LIN {X 0,Y 328.389,Z 347.877,A -85,B 0,C 180,E1 -14879.488,E2 -14879.488} C_VEL
LIN {X 0,Y 329.533,Z 341.284,A -85,B 0,C 180,E1 -14882.946,E2 -14882.946} C_VEL
LIN {X 0,Y 330.904,Z 335.131,A -85,B 0,C 180,E1 -14886.49,E2 -14886.49} C_VEL
LIN {X 0,Y 331.138,Z 332.463,A -85,B 0,C 180,E1 -14888.253,E2 -14888.253} C_VEL
LIN {X 0,Y 330.484,Z 328.715,A -85,B 0,C 180,E1 -14891.242,E2 -14891.242} C_VEL
LIN {X 0,Y 329.857,Z 325.225,A -85,B 0,C 180,E1 -14894.677,E2 -14894.677} C_VEL
LIN {X 0,Y 329.364,Z 322.49,A -85,B 0,C 180,E1 -14898.317,E2 -14898.317} C_VEL
LIN {X 0,Y 329.011,Z 320.792,A -85,B 0,C 180,E1 -14901.723,E2 -14901.723} C_VEL
LIN {X 0,Y 328.795,Z 319.94,A -85,B 0,C 180,E1 -14904.751,E2 -14904.751} C_VEL
LIN {X 0,Y 328.622,Z 319.641,A -85,B 0,C 180,E1 -14907.679,E2 -14907.679} C_VEL
LIN {X 0,Y 328.631,Z 319.835,A -85,B 0,C 180,E1 -14911.261,E2 -14911.261} C_VEL
LIN {X 0,Y 328.579,Z 320.736,A -85,B 0,C 180,E1 -14914.803,E2 -14914.803} C_VEL
LIN {X 0,Y 329.786,Z 323.377,A -85,B 0,C 180,E1 -14915.189,E2 -14915.189} C_VEL
LIN {X 0,Y 331.608,Z 326.284,A -85,B 0,C 180,E1 -14915.69,E2 -14915.69} C_VEL
LIN {X 0,Y 336.582,Z 336.57,A -85,B 0,C 180,E1 -14917.291,E2 -14917.291} C_VEL
LIN {X 0,Y 339.409,Z 344.725,A -85,B 0,C 180,E1 -14918.474,E2 -14918.474} C_VEL
LIN {X 0,Y 339.579,Z 346.937,A -85,B 0,C 180,E1 -14918.735,E2 -14918.735} C_VEL
LIN {X 0,Y 338.027,Z 357.85,A -85,B 0,C 180,E1 -14919.853,E2 -14919.853} C_VEL
LIN {X 0,Y 336.397,Z 367.772,A -85,B 0,C 180,E1 -14921.106,E2 -14921.106} C_VEL
LIN {X 0,Y 334.71,Z 377.405,A -85,B 0,C 180,E1 -14922.59,E2 -14922.59} C_VEL
LIN {X 0,Y 333.131,Z 385.421,A -85,B 0,C 180,E1 -14924.082,E2 -14924.082} C_VEL
LIN {X 0,Y 331.535,Z 393.277,A -85,B 0,C 180,E1 -14925.89,E2 -14925.89} C_VEL
LIN {X 0,Y 330.035,Z 399.65,A -85,B 0,C 180,E1 -14927.705,E2 -14927.705} C_VEL
LIN {X 0,Y 328.96,Z 404.549,A -85,B 0,C 180,E1 -14929.49,E2 -14929.49} C_VEL
LIN {X 0,Y 327.87,Z 408.533,A -85,B 0,C 180,E1 -14931.37,E2 -14931.37} C_VEL
LIN {X 0,Y 327.396,Z 410.536,A -85,B 0,C 180,E1 -14932.6,E2 -14932.6} C_VEL
LIN {X 0,Y 326.97,Z 412.06,A -85,B 0,C 180,E1 -14933.83,E2 -14933.83} C_VEL
LIN {X 0,Y 326.554,Z 413.149,A -85,B 0,C 180,E1 -14935.062,E2 -14935.062} C_VEL
LIN {X 0,Y 326.145,Z 413.838,A -85,B 0,C 180,E1 -14936.294,E2 -14936.294} C_VEL
LIN {X 0,Y 325.84,Z 414.097,A -85,B 0,C 180,E1 -14937.528,E2 -14937.528} C_VEL
LIN {X 0,Y 325.67,Z 413.896,A -85,B 0,C 180,E1 -14938.764,E2 -14938.764} C_VEL
LIN {X 0,Y 325.61,Z 413.286,A -85,B 0,C 180,E1 -14940,E2 -14940} C_VEL
LIN {X 0,Y 325.631,Z 412.265,A -85,B 0,C 180,E1 -14941.237,E2 -14941.237} C_VEL
LIN {X 0,Y 325.654,Z 410.778,A -85,B 0,C 180,E1 -14942.474,E2 -14942.474} C_VEL
LIN {X 0,Y 325.946,Z 407.724,A -85,B 0,C 180,E1 -14944.328,E2 -14944.328} C_VEL
LIN {X 0,Y 326.069,Z 403.613,A -85,B 0,C 180,E1 -14946.187,E2 -14946.187} C_VEL
LIN {X 0,Y 326.438,Z 397.331,A -85,B 0,C 180,E1 -14948.356,E2 -14948.356} C_VEL
LIN {X 0,Y 326.972,Z 390.471,A -85,B 0,C 180,E1 -14950.214,E2 -14950.214} C_VEL
LIN {X 0,Y 327.683,Z 381.942,A -85,B 0,C 180,E1 -14952.071,E2 -14952.071} C_VEL
LIN {X 0,Y 328.388,Z 373.312,A -85,B 0,C 180,E1 -14953.616,E2 -14953.616} C_VEL
LIN {X 0,Y 329.324,Z 362.847,A -85,B 0,C 180,E1 -14955.155,E2 -14955.155} C_VEL
LIN {X 0,Y 330.164,Z 350.596,A -85,B 0,C 180,E1 -14956.613,E2 -14956.613} C_VEL
LIN {X 0,Y 330.93,Z 338.24,A -85,B 0,C 180,E1 -14957.775,E2 -14957.775} C_VEL
LIN {X 0,Y 331.318,Z 331.336,A -85,B 0,C 180,E1 -14958.313,E2 -14958.313} C_VEL
LIN {X 0,Y 328.408,Z 318.06,A -85,B 0,C 180,E1 -14959.286,E2 -14959.286} C_VEL
LIN {X 0,Y 326.112,Z 308.863,A -85,B 0,C 180,E1 -14959.869,E2 -14959.869} C_VEL
LIN {X 0,Y 326.351,Z 308.833,A -85,B 0,C 180,E1 -14962.807,E2 -14962.807} C_VEL
LIN {X 0,Y 326.567,Z 308.8,A -85,B 0,C 180,E1 -14965.494,E2 -14965.494} C_VEL
LIN {X 0,Y 326.634,Z 308.796,A -85,B 0,C 180,E1 -14968.253,E2 -14968.253} C_VEL
LIN {X 0,Y 326.592,Z 308.795,A -85,B 0,C 180,E1 -14971.095,E2 -14971.095} C_VEL
LIN {X 0,Y 326.61,Z 308.804,A -85,B 0,C 180,E1 -14974.019,E2 -14974.019} C_VEL
LIN {X 0,Y 326.63,Z 308.801,A -85,B 0,C 180,E1 -14977.239,E2 -14977.239} C_VEL
LIN {X 0,Y 326.58,Z 308.807,A -85,B 0,C 180,E1 -14981.131,E2 -14981.131} C_VEL
LIN {X 0,Y 326.53,Z 308.809,A -85,B 0,C 180,E1 -14984.743,E2 -14984.743} C_VEL
LIN {X 0,Y 326.578,Z 308.805,A -85,B 0,C 180,E1 -14988.154,E2 -14988.154} C_VEL
LIN {X 0,Y 326.598,Z 308.804,A -85,B 0,C 180,E1 -14991.388,E2 -14991.388} C_VEL
LIN {X 0,Y 326.571,Z 308.814,A -85,B 0,C 180,E1 -14994.598,E2 -14994.598} C_VEL
LIN {X 0,Y 326.816,Z 310.846,A -85,B 0,C 180,E1 -14996.005,E2 -14996.005} C_VEL
LIN {X 0,Y 326.471,Z 317.34,A -85,B 0,C 180,E1 -15000.322,E2 -15000.322} C_VEL
LIN {X 0,Y 326.342,Z 322.733,A -85,B 0,C 180,E1 -15003.801,E2 -15003.801} C_VEL
LIN {X 0,Y 326.339,Z 329.269,A -85,B 0,C 180,E1 -15007.772,E2 -15007.772} C_VEL
LIN {X 0,Y 330.703,Z 344.202,A -85,B 0,C 180,E1 -15008.694,E2 -15008.694} C_VEL
LIN {X 0,Y 333.363,Z 356.048,A -85,B 0,C 180,E1 -15009.607,E2 -15009.607} C_VEL
LIN {X 0,Y 334.3,Z 361.022,A -85,B 0,C 180,E1 -15010.049,E2 -15010.049} C_VEL
LIN {X 0,Y 333.305,Z 372.846,A -85,B 0,C 180,E1 -15011.083,E2 -15011.083} C_VEL
LIN {X 0,Y 332.083,Z 384.217,A -85,B 0,C 180,E1 -15012.355,E2 -15012.355} C_VEL
LIN {X 0,Y 331.074,Z 393.497,A -85,B 0,C 180,E1 -15013.664,E2 -15013.664} C_VEL
LIN {X 0,Y 329.738,Z 402.364,A -85,B 0,C 180,E1 -15015.181,E2 -15015.181} C_VEL
LIN {X 0,Y 328.555,Z 410.995,A -85,B 0,C 180,E1 -15017.02,E2 -15017.02} C_VEL
LIN {X 0,Y 327.501,Z 417.914,A -85,B 0,C 180,E1 -15018.864,E2 -15018.864} C_VEL
LIN {X 0,Y 326.701,Z 423.408,A -85,B 0,C 180,E1 -15020.715,E2 -15020.715} C_VEL
LIN {X 0,Y 326.02,Z 428.45,A -85,B 0,C 180,E1 -15022.946,E2 -15022.946} C_VEL
LIN {X 0,Y 325.518,Z 431.838,A -85,B 0,C 180,E1 -15025.046,E2 -15025.046} C_VEL
LIN {X 0,Y 325.427,Z 433.241,A -85,B 0,C 180,E1 -15026.285,E2 -15026.285} C_VEL
LIN {X 0,Y 325.344,Z 434.228,A -85,B 0,C 180,E1 -15027.524,E2 -15027.524} C_VEL
LIN {X 0,Y 325.209,Z 435.072,A -85,B 0,C 180,E1 -15030,E2 -15030} C_VEL
LIN {X 0,Y 325.34,Z 434.294,A -85,B 0,C 180,E1 -15032.476,E2 -15032.476} C_VEL
LIN {X 0,Y 325.404,Z 433.335,A -85,B 0,C 180,E1 -15033.715,E2 -15033.715} C_VEL
LIN {X 0,Y 325.498,Z 431.982,A -85,B 0,C 180,E1 -15034.955,E2 -15034.955} C_VEL
LIN {X 0,Y 325.994,Z 428.727,A -85,B 0,C 180,E1 -15037.017,E2 -15037.017} C_VEL
LIN {X 0,Y 326.626,Z 423.679,A -85,B 0,C 180,E1 -15039.287,E2 -15039.287} C_VEL
LIN {X 0,Y 327.463,Z 418.244,A -85,B 0,C 180,E1 -15041.137,E2 -15041.137} C_VEL
LIN {X 0,Y 328.501,Z 411.435,A -85,B 0,C 180,E1 -15042.982,E2 -15042.982} C_VEL
LIN {X 0,Y 329.698,Z 402.902,A -85,B 0,C 180,E1 -15044.821,E2 -15044.821} C_VEL
LIN {X 0,Y 331.04,Z 394.145,A -85,B 0,C 180,E1 -15046.338,E2 -15046.338} C_VEL
LIN {X 0,Y 332.114,Z 384.041,A -85,B 0,C 180,E1 -15047.774,E2 -15047.774} C_VEL
LIN {X 0,Y 333.36,Z 372.347,A -85,B 0,C 180,E1 -15049.073,E2 -15049.073} C_VEL
LIN {X 0,Y 334.401,Z 361.794,A -85,B 0,C 180,E1 -15049.987,E2 -15049.987} C_VEL
LIN {X 0,Y 332.363,Z 351.218,A -85,B 0,C 180,E1 -15050.895,E2 -15050.895} C_VEL
LIN {X 0,Y 329.213,Z 338.732,A -85,B 0,C 180,E1 -15051.777,E2 -15051.777} C_VEL
LIN {X 0,Y 326.37,Z 329.318,A -85,B 0,C 180,E1 -15052.32,E2 -15052.32} C_VEL
LIN {X 0,Y 326.345,Z 322.926,A -85,B 0,C 180,E1 -15056.198,E2 -15056.198} C_VEL
LIN {X 0,Y 326.48,Z 317.517,A -85,B 0,C 180,E1 -15059.677,E2 -15059.677} C_VEL
LIN {X 0,Y 326.824,Z 311.012,A -85,B 0,C 180,E1 -15063.994,E2 -15063.994} C_VEL
LIN {X 0,Y 326.594,Z 308.806,A -85,B 0,C 180,E1 -15065.522,E2 -15065.522} C_VEL
LIN {X 0,Y 326.613,Z 308.802,A -85,B 0,C 180,E1 -15069.227,E2 -15069.227} C_VEL
LIN {X 0,Y 326.578,Z 308.809,A -85,B 0,C 180,E1 -15072.972,E2 -15072.972} C_VEL
LIN {X 0,Y 326.578,Z 308.807,A -85,B 0,C 180,E1 -15077.028,E2 -15077.028} C_VEL
LIN {X 0,Y 326.612,Z 308.801,A -85,B 0,C 180,E1 -15080.773,E2 -15080.773} C_VEL
LIN {X 0,Y 326.528,Z 308.807,A -85,B 0,C 180,E1 -15083.972,E2 -15083.972} C_VEL
LIN {X 0,Y 325.824,Z 309.013,A -85,B 0,C 180,E1 -15084.998,E2 -15084.998} C_VEL
LIN {X 0,Y 324.191,Z 309.573,A -85,B 0,C 180,E1 -15086,E2 -15086} C_VEL
LIN {X 0,Y 320.337,Z 311.597,A -85,B 0,C 180,E1 -15087.986,E2 -15087.986} C_VEL
LIN {X 0,Y 319.2,Z 313.002,A -85,B 0,C 180,E1 -15089.007,E2 -15089.007} C_VEL
LIN {X 0,Y 319.08,Z 313.52,A -85,B 0,C 180,E1 -15089.351,E2 -15089.351} C_VEL
LIN {X 0,Y 318.923,Z 319.269,A -85,B 0,C 180,E1 -15093.144,E2 -15093.144} C_VEL
LIN {X 0,Y 318.828,Z 324.595,A -85,B 0,C 180,E1 -15096.623,E2 -15096.623} C_VEL
LIN {X 0,Y 318.728,Z 329.745,A -85,B 0,C 180,E1 -15099.955,E2 -15099.955} C_VEL
LIN {X 0,Y 321.159,Z 342.779,A -85,B 0,C 180,E1 -15100.685,E2 -15100.685} C_VEL
LIN {X 0,Y 323.621,Z 355.679,A -85,B 0,C 180,E1 -15101.649,E2 -15101.649} C_VEL
LIN {X 0,Y 323.48,Z 361.623,A -85,B 0,C 180,E1 -15102.129,E2 -15102.129} C_VEL
LIN {X 0,Y 322.624,Z 373.758,A -85,B 0,C 180,E1 -15103.285,E2 -15103.285} C_VEL
LIN {X 0,Y 321.819,Z 385.197,A -85,B 0,C 180,E1 -15104.652,E2 -15104.652} C_VEL
LIN {X 0,Y 320.97,Z 394.854,A -85,B 0,C 180,E1 -15106.063,E2 -15106.063} C_VEL
LIN {X 0,Y 320.061,Z 405.398,A -85,B 0,C 180,E1 -15107.959,E2 -15107.959} C_VEL
LIN {X 0,Y 319.336,Z 413.85,A -85,B 0,C 180,E1 -15109.859,E2 -15109.859} C_VEL
LIN {X 0,Y 318.801,Z 420.704,A -85,B 0,C 180,E1 -15111.761,E2 -15111.761} C_VEL
LIN {X 0,Y 318.416,Z 426.181,A -85,B 0,C 180,E1 -15113.664,E2 -15113.664} C_VEL
LIN {X 0,Y 318.282,Z 430.405,A -85,B 0,C 180,E1 -15115.567,E2 -15115.567} C_VEL
LIN {X 0,Y 318.126,Z 433.53,A -85,B 0,C 180,E1 -15117.468,E2 -15117.468} C_VEL
LIN {X 0,Y 318.112,Z 435.035,A -85,B 0,C 180,E1 -15118.734,E2 -15118.734} C_VEL
LIN {X 0,Y 318.172,Z 436.12,A -85,B 0,C 180,E1 -15120,E2 -15120} C_VEL
LIN {X 0,Y 318.254,Z 436.733,A -85,B 0,C 180,E1 -15121.265,E2 -15121.265} C_VEL
LIN {X 0,Y 318.421,Z 436.924,A -85,B 0,C 180,E1 -15122.53,E2 -15122.53} C_VEL
LIN {X 0,Y 318.669,Z 436.708,A -85,B 0,C 180,E1 -15123.794,E2 -15123.794} C_VEL
LIN {X 0,Y 318.948,Z 436.024,A -85,B 0,C 180,E1 -15125.057,E2 -15125.057} C_VEL
LIN {X 0,Y 319.369,Z 433.443,A -85,B 0,C 180,E1 -15127.587,E2 -15127.587} C_VEL
LIN {X 0,Y 320.376,Z 430.263,A -85,B 0,C 180,E1 -15129.47,E2 -15129.47} C_VEL
LIN {X 0,Y 321.316,Z 425.996,A -85,B 0,C 180,E1 -15131.353,E2 -15131.353} C_VEL
LIN {X 0,Y 322.763,Z 419.488,A -85,B 0,C 180,E1 -15133.537,E2 -15133.537} C_VEL
LIN {X 0,Y 324.353,Z 412.416,A -85,B 0,C 180,E1 -15135.392,E2 -15135.392} C_VEL
LIN {X 0,Y 326.182,Z 403.606,A -85,B 0,C 180,E1 -15137.233,E2 -15137.233} C_VEL
LIN {X 0,Y 328.209,Z 393.435,A -85,B 0,C 180,E1 -15138.95,E2 -15138.95} C_VEL
LIN {X 0,Y 330.118,Z 382.681,A -85,B 0,C 180,E1 -15140.419,E2 -15140.419} C_VEL
LIN {X 0,Y 332.217,Z 369.516,A -85,B 0,C 180,E1 -15141.838,E2 -15141.838} C_VEL
LIN {X 0,Y 332.351,Z 368.078,A -85,B 0,C 180,E1 -15141.981,E2 -15141.981} C_VEL
LIN {X 0,Y 330.162,Z 358.055,A -85,B 0,C 180,E1 -15143.305,E2 -15143.305} C_VEL
LIN {X 0,Y 326.236,Z 347.061,A -85,B 0,C 180,E1 -15144.856,E2 -15144.856} C_VEL
LIN {X 0,Y 323.056,Z 340.093,A -85,B 0,C 180,E1 -15145.906,E2 -15145.906} C_VEL
LIN {X 0,Y 321.796,Z 337.014,A -85,B 0,C 180,E1 -15146.354,E2 -15146.354} C_VEL
LIN {X 0,Y 322.533,Z 332.112,A -85,B 0,C 180,E1 -15150.078,E2 -15150.078} C_VEL
LIN {X 0,Y 323.218,Z 328.529,A -85,B 0,C 180,E1 -15152.929,E2 -15152.929} C_VEL
LIN {X 0,Y 323.383,Z 326.836,A -85,B 0,C 180,E1 -15154.406,E2 -15154.406} C_VEL
LIN {X 0,Y 323.298,Z 324.738,A -85,B 0,C 180,E1 -15156.455,E2 -15156.455} C_VEL
LIN {X 0,Y 323.004,Z 322.421,A -85,B 0,C 180,E1 -15159.123,E2 -15159.123} C_VEL
LIN {X 0,Y 322.6,Z 320.404,A -85,B 0,C 180,E1 -15162.208,E2 -15162.208} C_VEL
LIN {X 0,Y 322.049,Z 319.739,A -85,B 0,C 180,E1 -15164.293,E2 -15164.293} C_VEL
LIN {X 0,Y 321.458,Z 319.688,A -85,B 0,C 180,E1 -15166.547,E2 -15166.547} C_VEL
LIN {X 0,Y 322.812,Z 326.631,A -85,B 0,C 180,E1 -15170.285,E2 -15170.285} C_VEL
LIN {X 0,Y 323.47,Z 330.981,A -85,B 0,C 180,E1 -15172.529,E2 -15172.529} C_VEL
LIN {X 0,Y 322.945,Z 335.629,A -85,B 0,C 180,E1 -15174.781,E2 -15174.781} C_VEL
LIN {X 0,Y 321.872,Z 343.274,A -85,B 0,C 180,E1 -15178.397,E2 -15178.397} C_VEL
LIN {X 0,Y 320.746,Z 352.365,A -85,B 0,C 180,E1 -15182.604,E2 -15182.604} C_VEL
LIN {X 0,Y 320.405,Z 355.766,A -85,B 0,C 180,E1 -15184.07,E2 -15184.07} C_VEL
LIN {X 0,Y 321.285,Z 359.893,A -85,B 0,C 180,E1 -15184.469,E2 -15184.469} C_VEL
LIN {X 0,Y 321.976,Z 362.193,A -85,B 0,C 180,E1 -15184.716,E2 -15184.716} C_VEL
LIN {X 0,Y 324.913,Z 374.79,A -85,B 0,C 180,E1 -15185.952,E2 -15185.952} C_VEL
LIN {X 0,Y 326.631,Z 386.508,A -85,B 0,C 180,E1 -15187.1,E2 -15187.1} C_VEL
LIN {X 0,Y 326.814,Z 401.047,A -85,B 0,C 180,E1 -15188.557,E2 -15188.557} C_VEL
LIN {X 0,Y 326.653,Z 413.267,A -85,B 0,C 180,E1 -15190.028,E2 -15190.028} C_VEL
LIN {X 0,Y 324.612,Z 424.833,A -85,B 0,C 180,E1 -15191.54,E2 -15191.54} C_VEL
LIN {X 0,Y 322.759,Z 435.331,A -85,B 0,C 180,E1 -15193.264,E2 -15193.264} C_VEL
LIN {X 0,Y 321.272,Z 444.462,A -85,B 0,C 180,E1 -15195.106,E2 -15195.106} C_VEL
LIN {X 0,Y 320.021,Z 452.055,A -85,B 0,C 180,E1 -15196.991,E2 -15196.991} C_VEL
LIN {X 0,Y 319.016,Z 459.185,A -85,B 0,C 180,E1 -15199.207,E2 -15199.207} C_VEL
LIN {X 0,Y 318.414,Z 464.012,A -85,B 0,C 180,E1 -15201.112,E2 -15201.112} C_VEL
LIN {X 0,Y 318.142,Z 467.739,A -85,B 0,C 180,E1 -15203.021,E2 -15203.021} C_VEL
LIN {X 0,Y 317.959,Z 470.454,A -85,B 0,C 180,E1 -15204.928,E2 -15204.928} C_VEL
LIN {X 0,Y 317.981,Z 471.724,A -85,B 0,C 180,E1 -15206.198,E2 -15206.198} C_VEL
LIN {X 0,Y 318.095,Z 472.979,A -85,B 0,C 180,E1 -15208.734,E2 -15208.734} C_VEL
LIN {X 0,Y 318.215,Z 472.983,A -85,B 0,C 180,E1 -15210,E2 -15210} C_VEL
LIN {X 0,Y 317.968,Z 471.876,A -85,B 0,C 180,E1 -15212.534,E2 -15212.534} C_VEL
LIN {X 0,Y 317.985,Z 470.852,A -85,B 0,C 180,E1 -15213.802,E2 -15213.802} C_VEL
LIN {X 0,Y 318.114,Z 467.745,A -85,B 0,C 180,E1 -15216.187,E2 -15216.187} C_VEL
LIN {X 0,Y 318.273,Z 463.753,A -85,B 0,C 180,E1 -15218.252,E2 -15218.252} C_VEL
LIN {X 0,Y 318.728,Z 458.888,A -85,B 0,C 180,E1 -15220.16,E2 -15220.16} C_VEL
LIN {X 0,Y 319.953,Z 449.69,A -85,B 0,C 180,E1 -15223.012,E2 -15223.012} C_VEL
LIN {X 0,Y 321.346,Z 440.86,A -85,B 0,C 180,E1 -15225.215,E2 -15225.215} C_VEL
LIN {X 0,Y 322.877,Z 431.604,A -85,B 0,C 180,E1 -15227.089,E2 -15227.089} C_VEL
LIN {X 0,Y 325.018,Z 420.298,A -85,B 0,C 180,E1 -15228.926,E2 -15228.926} C_VEL
LIN {X 0,Y 326.586,Z 411.332,A -85,B 0,C 180,E1 -15230.14,E2 -15230.14} C_VEL
LIN {X 0,Y 326.871,Z 400.124,A -85,B 0,C 180,E1 -15231.564,E2 -15231.564} C_VEL
LIN {X 0,Y 326.921,Z 389.197,A -85,B 0,C 180,E1 -15232.765,E2 -15232.765} C_VEL
LIN {X 0,Y 325.801,Z 378.126,A -85,B 0,C 180,E1 -15233.943,E2 -15233.943} C_VEL
LIN {X 0,Y 323.834,Z 367.884,A -85,B 0,C 180,E1 -15235.031,E2 -15235.031} C_VEL
LIN {X 0,Y 321.496,Z 359.207,A -85,B 0,C 180,E1 -15235.986,E2 -15235.986} C_VEL
LIN {X 0,Y 320.514,Z 355.252,A -85,B 0,C 180,E1 -15236.422,E2 -15236.422} C_VEL
LIN {X 0,Y 321.598,Z 347.856,A -85,B 0,C 180,E1 -15240.174,E2 -15240.174} C_VEL
LIN {X 0,Y 322.769,Z 341.576,A -85,B 0,C 180,E1 -15243.617,E2 -15243.617} C_VEL
LIN {X 0,Y 323.987,Z 336.568,A -85,B 0,C 180,E1 -15246.62,E2 -15246.62} C_VEL
LIN {X 0,Y 324.144,Z 333.59,A -85,B 0,C 180,E1 -15248.689,E2 -15248.689} C_VEL
LIN {X 0,Y 323.757,Z 331.199,A -85,B 0,C 180,E1 -15250.635,E2 -15250.635} C_VEL
LIN {X 0,Y 323.088,Z 327.59,A -85,B 0,C 180,E1 -15254.124,E2 -15254.124} C_VEL
LIN {X 0,Y 322.546,Z 324.723,A -85,B 0,C 180,E1 -15257.803,E2 -15257.803} C_VEL
LIN {X 0,Y 322.233,Z 323.095,A -85,B 0,C 180,E1 -15260.765,E2 -15260.765} C_VEL
LIN {X 0,Y 321.983,Z 322.01,A -85,B 0,C 180,E1 -15263.89,E2 -15263.89} C_VEL
LIN {X 0,Y 321.799,Z 321.521,A -85,B 0,C 180,E1 -15266.907,E2 -15266.907} C_VEL
LIN {X 0,Y 321.751,Z 321.57,A -85,B 0,C 180,E1 -15270.894,E2 -15270.894} C_VEL
LIN {X 0,Y 321.782,Z 322.229,A -85,B 0,C 180,E1 -15273.719,E2 -15273.719} C_VEL
LIN {X 0,Y 322.426,Z 323.833,A -85,B 0,C 180,E1 -15273.953,E2 -15273.953} C_VEL
LIN {X 0,Y 325.754,Z 329.118,A -85,B 0,C 180,E1 -15274.977,E2 -15274.977} C_VEL
LIN {X 0,Y 330.414,Z 338.603,A -85,B 0,C 180,E1 -15276.6,E2 -15276.6} C_VEL
LIN {X 0,Y 333.262,Z 346.705,A -85,B 0,C 180,E1 -15277.864,E2 -15277.864} C_VEL
LIN {X 0,Y 333.641,Z 348.636,A -85,B 0,C 180,E1 -15278.139,E2 -15278.139} C_VEL
LIN {X 0,Y 331.8,Z 360.17,A -85,B 0,C 180,E1 -15279.382,E2 -15279.382} C_VEL
LIN {X 0,Y 329.855,Z 371.32,A -85,B 0,C 180,E1 -15280.878,E2 -15280.878} C_VEL
LIN {X 0,Y 327.88,Z 381.241,A -85,B 0,C 180,E1 -15282.537,E2 -15282.537} C_VEL
LIN {X 0,Y 325.951,Z 390.069,A -85,B 0,C 180,E1 -15284.364,E2 -15284.364} C_VEL
LIN {X 0,Y 324.316,Z 397.189,A -85,B 0,C 180,E1 -15286.21,E2 -15286.21} C_VEL
LIN {X 0,Y 322.913,Z 402.85,A -85,B 0,C 180,E1 -15288.067,E2 -15288.067} C_VEL
LIN {X 0,Y 321.667,Z 407.357,A -85,B 0,C 180,E1 -15289.934,E2 -15289.934} C_VEL
LIN {X 0,Y 320.982,Z 409.734,A -85,B 0,C 180,E1 -15291.184,E2 -15291.184} C_VEL
LIN {X 0,Y 320.446,Z 411.634,A -85,B 0,C 180,E1 -15292.438,E2 -15292.438} C_VEL
LIN {X 0,Y 319.985,Z 413.053,A -85,B 0,C 180,E1 -15293.695,E2 -15293.695} C_VEL
LIN {X 0,Y 319.547,Z 414.078,A -85,B 0,C 180,E1 -15294.953,E2 -15294.953} C_VEL
LIN {X 0,Y 319.123,Z 414.704,A -85,B 0,C 180,E1 -15296.212,E2 -15296.212} C_VEL
LIN {X 0,Y 318.806,Z 414.862,A -85,B 0,C 180,E1 -15297.473,E2 -15297.473} C_VEL
LIN {X 0,Y 318.628,Z 414.6,A -85,B 0,C 180,E1 -15298.736,E2 -15298.736} C_VEL
LIN {X 0,Y 318.565,Z 413.925,A -85,B 0,C 180,E1 -15300,E2 -15300} C_VEL
LIN {X 0,Y 318.556,Z 412.809,A -85,B 0,C 180,E1 -15301.264,E2 -15301.264} C_VEL
LIN {X 0,Y 318.595,Z 411.251,A -85,B 0,C 180,E1 -15302.529,E2 -15302.529} C_VEL
LIN {X 0,Y 318.898,Z 408.081,A -85,B 0,C 180,E1 -15304.424,E2 -15304.424} C_VEL
LIN {X 0,Y 319.023,Z 403.842,A -85,B 0,C 180,E1 -15306.324,E2 -15306.324} C_VEL
LIN {X 0,Y 319.4,Z 397.393,A -85,B 0,C 180,E1 -15308.541,E2 -15308.541} C_VEL
LIN {X 0,Y 319.961,Z 390.334,A -85,B 0,C 180,E1 -15310.441,E2 -15310.441} C_VEL
LIN {X 0,Y 320.704,Z 381.653,A -85,B 0,C 180,E1 -15312.337,E2 -15312.337} C_VEL
LIN {X 0,Y 321.533,Z 371.847,A -85,B 0,C 180,E1 -15314.074,E2 -15314.074} C_VEL
LIN {X 0,Y 322.52,Z 360.943,A -85,B 0,C 180,E1 -15315.644,E2 -15315.644} C_VEL
LIN {X 0,Y 323.351,Z 348.84,A -85,B 0,C 180,E1 -15317.05,E2 -15317.05} C_VEL
LIN {X 0,Y 324.11,Z 336.798,A -85,B 0,C 180,E1 -15318.162,E2 -15318.162} C_VEL
LIN {X 0,Y 324.277,Z 331.719,A -85,B 0,C 180,E1 -15318.561,E2 -15318.561} C_VEL
LIN {X 0,Y 321.294,Z 318.441,A -85,B 0,C 180,E1 -15319.559,E2 -15319.559} C_VEL
LIN {X 0,Y 319.097,Z 309.735,A -85,B 0,C 180,E1 -15320.129,E2 -15320.129} C_VEL
LIN {X 0,Y 319.342,Z 309.707,A -85,B 0,C 180,E1 -15323.337,E2 -15323.337} C_VEL
LIN {X 0,Y 319.541,Z 309.674,A -85,B 0,C 180,E1 -15326.097,E2 -15326.097} C_VEL
LIN {X 0,Y 319.571,Z 309.678,A -85,B 0,C 180,E1 -15328.936,E2 -15328.936} C_VEL
LIN {X 0,Y 319.534,Z 309.676,A -85,B 0,C 180,E1 -15331.862,E2 -15331.862} C_VEL
LIN {X 0,Y 319.582,Z 309.67,A -85,B 0,C 180,E1 -15335.543,E2 -15335.543} C_VEL
LIN {X 0,Y 319.575,Z 309.68,A -85,B 0,C 180,E1 -15338.008,E2 -15338.008} C_VEL
LIN {X 0,Y 319.528,Z 309.685,A -85,B 0,C 180,E1 -15341.597,E2 -15341.597} C_VEL
LIN {X 0,Y 319.491,Z 309.687,A -85,B 0,C 180,E1 -15345.257,E2 -15345.257} C_VEL
LIN {X 0,Y 319.53,Z 309.682,A -85,B 0,C 180,E1 -15348.712,E2 -15348.712} C_VEL
LIN {X 0,Y 319.547,Z 309.682,A -85,B 0,C 180,E1 -15352.352,E2 -15352.352} C_VEL
LIN {X 0,Y 319.54,Z 309.735,A -85,B 0,C 180,E1 -15354.327,E2 -15354.327} C_VEL
LIN {X 0,Y 319.833,Z 312.003,A -85,B 0,C 180,E1 -15355.921,E2 -15355.921} C_VEL
LIN {X 0,Y 319.472,Z 318.605,A -85,B 0,C 180,E1 -15360.332,E2 -15360.332} C_VEL
LIN {X 0,Y 319.367,Z 324.117,A -85,B 0,C 180,E1 -15363.888,E2 -15363.888} C_VEL
LIN {X 0,Y 319.366,Z 329.79,A -85,B 0,C 180,E1 -15367.286,E2 -15367.286} C_VEL
LIN {X 0,Y 323.359,Z 343.157,A -85,B 0,C 180,E1 -15368.114,E2 -15368.114} C_VEL
LIN {X 0,Y 326.094,Z 354.458,A -85,B 0,C 180,E1 -15368.988,E2 -15368.988} C_VEL
LIN {X 0,Y 327.607,Z 363.296,A -85,B 0,C 180,E1 -15369.785,E2 -15369.785} C_VEL
LIN {X 0,Y 326.46,Z 374.774,A -85,B 0,C 180,E1 -15370.834,E2 -15370.834} C_VEL
LIN {X 0,Y 325.295,Z 385.051,A -85,B 0,C 180,E1 -15372.032,E2 -15372.032} C_VEL
LIN {X 0,Y 324.021,Z 395.802,A -85,B 0,C 180,E1 -15373.622,E2 -15373.622} C_VEL
LIN {X 0,Y 322.693,Z 404.359,A -85,B 0,C 180,E1 -15375.173,E2 -15375.173} C_VEL
LIN {X 0,Y 321.456,Z 412.67,A -85,B 0,C 180,E1 -15377.05,E2 -15377.05} C_VEL
LIN {X 0,Y 320.565,Z 418.327,A -85,B 0,C 180,E1 -15378.62,E2 -15378.62} C_VEL
LIN {X 0,Y 319.69,Z 423.824,A -85,B 0,C 180,E1 -15380.51,E2 -15380.51} C_VEL
LIN {X 0,Y 318.954,Z 429.119,A -85,B 0,C 180,E1 -15382.923,E2 -15382.923} C_VEL
LIN {X 0,Y 318.465,Z 432.253,A -85,B 0,C 180,E1 -15384.936,E2 -15384.936} C_VEL
LIN {X 0,Y 318.346,Z 433.657,A -85,B 0,C 180,E1 -15386.203,E2 -15386.203} C_VEL
LIN {X 0,Y 318.26,Z 434.643,A -85,B 0,C 180,E1 -15387.469,E2 -15387.469} C_VEL
LIN {X 0,Y 318.134,Z 435.487,A -85,B 0,C 180,E1 -15390,E2 -15390} C_VEL
LIN {X 0,Y 318.16,Z 435.294,A -85,B 0,C 180,E1 -15391.266,E2 -15391.266} C_VEL
LIN {X 0,Y 318.255,Z 434.709,A -85,B 0,C 180,E1 -15392.531,E2 -15392.531} C_VEL
LIN {X 0,Y 318.323,Z 433.749,A -85,B 0,C 180,E1 -15393.798,E2 -15393.798} C_VEL
LIN {X 0,Y 318.447,Z 432.395,A -85,B 0,C 180,E1 -15395.065,E2 -15395.065} C_VEL
LIN {X 0,Y 318.929,Z 429.392,A -85,B 0,C 180,E1 -15397.04,E2 -15397.04} C_VEL
LIN {X 0,Y 319.431,Z 425.654,A -85,B 0,C 180,E1 -15398.86,E2 -15398.86} C_VEL
LIN {X 0,Y 320.17,Z 420.622,A -85,B 0,C 180,E1 -15400.753,E2 -15400.753} C_VEL
LIN {X 0,Y 321.223,Z 414.264,A -85,B 0,C 180,E1 -15402.638,E2 -15402.638} C_VEL
LIN {X 0,Y 322.417,Z 406.363,A -85,B 0,C 180,E1 -15404.518,E2 -15404.518} C_VEL
LIN {X 0,Y 323.69,Z 398.277,A -85,B 0,C 180,E1 -15406.071,E2 -15406.071} C_VEL
LIN {X 0,Y 324.966,Z 388.345,A -85,B 0,C 180,E1 -15407.625,E2 -15407.625} C_VEL
LIN {X 0,Y 326.237,Z 377.149,A -85,B 0,C 180,E1 -15409.016,E2 -15409.016} C_VEL
LIN {X 0,Y 327.382,Z 366.158,A -85,B 0,C 180,E1 -15410.089,E2 -15410.089} C_VEL
LIN {X 0,Y 327.651,Z 362.424,A -85,B 0,C 180,E1 -15410.396,E2 -15410.396} C_VEL
LIN {X 0,Y 325.194,Z 350.337,A -85,B 0,C 180,E1 -15411.462,E2 -15411.462} C_VEL
LIN {X 0,Y 321.765,Z 337.494,A -85,B 0,C 180,E1 -15412.373,E2 -15412.373} C_VEL
LIN {X 0,Y 319.355,Z 329.64,A -85,B 0,C 180,E1 -15412.858,E2 -15412.858} C_VEL
LIN {X 0,Y 319.384,Z 323.194,A -85,B 0,C 180,E1 -15416.814,E2 -15416.814} C_VEL
LIN {X 0,Y 319.507,Z 317.706,A -85,B 0,C 180,E1 -15420.392,E2 -15420.392} C_VEL
LIN {X 0,Y 319.845,Z 312.168,A -85,B 0,C 180,E1 -15424.077,E2 -15424.077} C_VEL
LIN {X 0,Y 319.54,Z 309.685,A -85,B 0,C 180,E1 -15425.929,E2 -15425.929} C_VEL
LIN {X 0,Y 319.56,Z 309.681,A -85,B 0,C 180,E1 -15429.669,E2 -15429.669} C_VEL
LIN {X 0,Y 319.524,Z 309.686,A -85,B 0,C 180,E1 -15433.461,E2 -15433.461} C_VEL
LIN {X 0,Y 319.556,Z 309.682,A -85,B 0,C 180,E1 -15437.017,E2 -15437.017} C_VEL
LIN {X 0,Y 319.548,Z 309.682,A -85,B 0,C 180,E1 -15440.371,E2 -15440.371} C_VEL
LIN {X 0,Y 319.5,Z 309.685,A -85,B 0,C 180,E1 -15443.966,E2 -15443.966} C_VEL
LIN {X 0,Y 319.35,Z 309.756,A -85,B 0,C 180,E1 -15446.868,E2 -15446.868} C_VEL
LIN {X 0,Y 319.08,Z 313.52,A -85,B 0,C 180,E1 -15449.351,E2 -15449.351} C_VEL
LIN {X 0,Y 318.337,Z 315.154,A -85,B 0,C 180,E1 -15450.363,E2 -15450.363} C_VEL
LIN {X 0,Y 315.435,Z 317.975,A -85,B 0,C 180,E1 -15452,E2 -15452} C_VEL
LIN {X 0,Y 312.995,Z 320.228,A -85,B 0,C 180,E1 -15453.326,E2 -15453.326} C_VEL
LIN {X 0,Y 311.92,Z 321.882,A -85,B 0,C 180,E1 -15454.356,E2 -15454.356} C_VEL
LIN {X 0,Y 311.816,Z 322.424,A -85,B 0,C 180,E1 -15454.706,E2 -15454.706} C_VEL
LIN {X 0,Y 311.75,Z 326.848,A -85,B 0,C 180,E1 -15457.562,E2 -15457.562} C_VEL
LIN {X 0,Y 311.706,Z 330.153,A -85,B 0,C 180,E1 -15459.696,E2 -15459.696} C_VEL
LIN {X 0,Y 314.303,Z 344.287,A -85,B 0,C 180,E1 -15460.522,E2 -15460.522} C_VEL
LIN {X 0,Y 316.608,Z 356.571,A -85,B 0,C 180,E1 -15461.471,E2 -15461.471} C_VEL
LIN {X 0,Y 316.426,Z 363.462,A -85,B 0,C 180,E1 -15462.051,E2 -15462.051} C_VEL
LIN {X 0,Y 315.462,Z 376.648,A -85,B 0,C 180,E1 -15463.393,E2 -15463.393} C_VEL
LIN {X 0,Y 314.641,Z 387.536,A -85,B 0,C 180,E1 -15464.784,E2 -15464.784} C_VEL
LIN {X 0,Y 313.681,Z 397.853,A -85,B 0,C 180,E1 -15466.393,E2 -15466.393} C_VEL
LIN {X 0,Y 312.954,Z 406.392,A -85,B 0,C 180,E1 -15468.011,E2 -15468.011} C_VEL
LIN {X 0,Y 312.226,Z 414.751,A -85,B 0,C 180,E1 -15469.953,E2 -15469.953} C_VEL
LIN {X 0,Y 311.687,Z 421.548,A -85,B 0,C 180,E1 -15471.898,E2 -15471.898} C_VEL
LIN {X 0,Y 311.351,Z 426.122,A -85,B 0,C 180,E1 -15473.52,E2 -15473.52} C_VEL
LIN {X 0,Y 311.218,Z 430.49,A -85,B 0,C 180,E1 -15475.467,E2 -15475.467} C_VEL
LIN {X 0,Y 311.036,Z 433.737,A -85,B 0,C 180,E1 -15477.41,E2 -15477.41} C_VEL
LIN {X 0,Y 311.017,Z 435.301,A -85,B 0,C 180,E1 -15478.705,E2 -15478.705} C_VEL
LIN {X 0,Y 311.08,Z 436.452,A -85,B 0,C 180,E1 -15480,E2 -15480} C_VEL
LIN {X 0,Y 311.181,Z 437.177,A -85,B 0,C 180,E1 -15481.294,E2 -15481.294} C_VEL
LIN {X 0,Y 311.355,Z 437.428,A -85,B 0,C 180,E1 -15482.587,E2 -15482.587} C_VEL
LIN {X 0,Y 311.615,Z 437.271,A -85,B 0,C 180,E1 -15483.88,E2 -15483.88} C_VEL
LIN {X 0,Y 311.923,Z 436.7,A -85,B 0,C 180,E1 -15485.171,E2 -15485.171} C_VEL
LIN {X 0,Y 312.073,Z 435.688,A -85,B 0,C 180,E1 -15486.465,E2 -15486.465} C_VEL
LIN {X 0,Y 312.383,Z 434.258,A -85,B 0,C 180,E1 -15487.758,E2 -15487.758} C_VEL
LIN {X 0,Y 313.446,Z 431.199,A -85,B 0,C 180,E1 -15489.681,E2 -15489.681} C_VEL
LIN {X 0,Y 314.461,Z 427.116,A -85,B 0,C 180,E1 -15491.604,E2 -15491.604} C_VEL
LIN {X 0,Y 315.986,Z 420.814,A -85,B 0,C 180,E1 -15493.833,E2 -15493.833} C_VEL
LIN {X 0,Y 317.667,Z 413.936,A -85,B 0,C 180,E1 -15495.725,E2 -15495.725} C_VEL
LIN {X 0,Y 319.606,Z 405.471,A -85,B 0,C 180,E1 -15497.599,E2 -15497.599} C_VEL
LIN {X 0,Y 321.848,Z 395.172,A -85,B 0,C 180,E1 -15499.415,E2 -15499.415} C_VEL
LIN {X 0,Y 324.083,Z 383.563,A -85,B 0,C 180,E1 -15501.064,E2 -15501.064} C_VEL
LIN {X 0,Y 326.305,Z 370.821,A -85,B 0,C 180,E1 -15502.476,E2 -15502.476} C_VEL
LIN {X 0,Y 324.863,Z 362.651,A -85,B 0,C 180,E1 -15503.615,E2 -15503.615} C_VEL
LIN {X 0,Y 320.937,Z 350.608,A -85,B 0,C 180,E1 -15505.426,E2 -15505.426} C_VEL
LIN {X 0,Y 316.778,Z 341.322,A -85,B 0,C 180,E1 -15506.954,E2 -15506.954} C_VEL
LIN {X 0,Y 315.258,Z 337.818,A -85,B 0,C 180,E1 -15507.543,E2 -15507.543} C_VEL
LIN {X 0,Y 316.01,Z 333.776,A -85,B 0,C 180,E1 -15510.765,E2 -15510.765} C_VEL
LIN {X 0,Y 316.68,Z 330.331,A -85,B 0,C 180,E1 -15513.698,E2 -15513.698} C_VEL
LIN {X 0,Y 316.793,Z 328.769,A -85,B 0,C 180,E1 -15515.226,E2 -15515.226} C_VEL
LIN {X 0,Y 316.738,Z 327.159,A -85,B 0,C 180,E1 -15516.985,E2 -15516.985} C_VEL
LIN {X 0,Y 316.518,Z 324.86,A -85,B 0,C 180,E1 -15520.085,E2 -15520.085} C_VEL
LIN {X 0,Y 316.178,Z 323.498,A -85,B 0,C 180,E1 -15522.817,E2 -15522.817} C_VEL
LIN {X 0,Y 315.505,Z 323.144,A -85,B 0,C 180,E1 -15525.464,E2 -15525.464} C_VEL
LIN {X 0,Y 315.029,Z 323.719,A -85,B 0,C 180,E1 -15528.086,E2 -15528.086} C_VEL
LIN {X 0,Y 316.243,Z 330.081,A -85,B 0,C 180,E1 -15531.519,E2 -15531.519} C_VEL
LIN {X 0,Y 316.364,Z 333.254,A -85,B 0,C 180,E1 -15533.144,E2 -15533.144} C_VEL
LIN {X 0,Y 315.218,Z 340.922,A -85,B 0,C 180,E1 -15536.89,E2 -15536.89} C_VEL
LIN {X 0,Y 314.094,Z 349.022,A -85,B 0,C 180,E1 -15540.767,E2 -15540.767} C_VEL
LIN {X 0,Y 313.643,Z 353.179,A -85,B 0,C 180,E1 -15542.7,E2 -15542.7} C_VEL
LIN {X 0,Y 314.357,Z 357.166,A -85,B 0,C 180,E1 -15543.114,E2 -15543.114} C_VEL
LIN {X 0,Y 315.349,Z 359.987,A -85,B 0,C 180,E1 -15543.481,E2 -15543.481} C_VEL
LIN {X 0,Y 318.337,Z 372.635,A -85,B 0,C 180,E1 -15544.846,E2 -15544.846} C_VEL
LIN {X 0,Y 320.411,Z 385.967,A -85,B 0,C 180,E1 -15546.256,E2 -15546.256} C_VEL
LIN {X 0,Y 320.6,Z 398.262,A -85,B 0,C 180,E1 -15547.544,E2 -15547.544} C_VEL
LIN {X 0,Y 320.408,Z 411.179,A -85,B 0,C 180,E1 -15549.118,E2 -15549.118} C_VEL
LIN {X 0,Y 320.123,Z 414.818,A -85,B 0,C 180,E1 -15549.603,E2 -15549.603} C_VEL
LIN {X 0,Y 318.148,Z 424.889,A -85,B 0,C 180,E1 -15550.984,E2 -15550.984} C_VEL
LIN {X 0,Y 316.027,Z 436.058,A -85,B 0,C 180,E1 -15552.896,E2 -15552.896} C_VEL
LIN {X 0,Y 314.432,Z 444.888,A -85,B 0,C 180,E1 -15554.774,E2 -15554.774} C_VEL
LIN {X 0,Y 312.885,Z 453.406,A -85,B 0,C 180,E1 -15557.019,E2 -15557.019} C_VEL
LIN {X 0,Y 312.005,Z 459.26,A -85,B 0,C 180,E1 -15558.962,E2 -15558.962} C_VEL
LIN {X 0,Y 311.382,Z 463.949,A -85,B 0,C 180,E1 -15560.91,E2 -15560.91} C_VEL
LIN {X 0,Y 310.989,Z 468.542,A -85,B 0,C 180,E1 -15563.512,E2 -15563.512} C_VEL
LIN {X 0,Y 310.873,Z 470.2,A -85,B 0,C 180,E1 -15564.812,E2 -15564.812} C_VEL
LIN {X 0,Y 310.905,Z 471.395,A -85,B 0,C 180,E1 -15566.111,E2 -15566.111} C_VEL
LIN {X 0,Y 310.997,Z 472.572,A -85,B 0,C 180,E1 -15568.705,E2 -15568.705} C_VEL
LIN {X 0,Y 311.154,Z 472.499,A -85,B 0,C 180,E1 -15570,E2 -15570} C_VEL
LIN {X 0,Y 310.881,Z 471.46,A -85,B 0,C 180,E1 -15572.591,E2 -15572.591} C_VEL
LIN {X 0,Y 310.913,Z 470.437,A -85,B 0,C 180,E1 -15573.888,E2 -15573.888} C_VEL
LIN {X 0,Y 311.039,Z 467.578,A -85,B 0,C 180,E1 -15576.178,E2 -15576.178} C_VEL
LIN {X 0,Y 311.224,Z 463.336,A -85,B 0,C 180,E1 -15578.441,E2 -15578.441} C_VEL
LIN {X 0,Y 311.694,Z 458.47,A -85,B 0,C 180,E1 -15580.392,E2 -15580.392} C_VEL
LIN {X 0,Y 313.017,Z 449.631,A -85,B 0,C 180,E1 -15583.305,E2 -15583.305} C_VEL
LIN {X 0,Y 314.22,Z 442.364,A -85,B 0,C 180,E1 -15585.237,E2 -15585.237} C_VEL
LIN {X 0,Y 316.127,Z 431.991,A -85,B 0,C 180,E1 -15587.465,E2 -15587.465} C_VEL
LIN {X 0,Y 318.15,Z 422.044,A -85,B 0,C 180,E1 -15589.183,E2 -15589.183} C_VEL
LIN {X 0,Y 319.996,Z 412.411,A -85,B 0,C 180,E1 -15590.573,E2 -15590.573} C_VEL
LIN {X 0,Y 320.507,Z 400.68,A -85,B 0,C 180,E1 -15592.142,E2 -15592.142} C_VEL
LIN {X 0,Y 320.649,Z 389.487,A -85,B 0,C 180,E1 -15593.451,E2 -15593.451} C_VEL
LIN {X 0,Y 319.376,Z 377.077,A -85,B 0,C 180,E1 -15594.874,E2 -15594.874} C_VEL
LIN {X 0,Y 316.755,Z 364.483,A -85,B 0,C 180,E1 -15596.344,E2 -15596.344} C_VEL
LIN {X 0,Y 314.876,Z 358.22,A -85,B 0,C 180,E1 -15597.13,E2 -15597.13} C_VEL
LIN {X 0,Y 313.819,Z 354.127,A -85,B 0,C 180,E1 -15597.613,E2 -15597.613} C_VEL
LIN {X 0,Y 315.043,Z 346.801,A -85,B 0,C 180,E1 -15601.492,E2 -15601.492} C_VEL
LIN {X 0,Y 316.44,Z 340.353,A -85,B 0,C 180,E1 -15605.271,E2 -15605.271} C_VEL
LIN {X 0,Y 317.157,Z 337.519,A -85,B 0,C 180,E1 -15607.085,E2 -15607.085} C_VEL
LIN {X 0,Y 317.179,Z 334.733,A -85,B 0,C 180,E1 -15609.147,E2 -15609.147} C_VEL
LIN {X 0,Y 316.439,Z 330.624,A -85,B 0,C 180,E1 -15612.868,E2 -15612.868} C_VEL
LIN {X 0,Y 315.866,Z 327.606,A -85,B 0,C 180,E1 -15616.39,E2 -15616.39} C_VEL
LIN {X 0,Y 315.503,Z 325.49,A -85,B 0,C 180,E1 -15619.76,E2 -15619.76} C_VEL
LIN {X 0,Y 315.178,Z 324.038,A -85,B 0,C 180,E1 -15623.394,E2 -15623.394} C_VEL
LIN {X 0,Y 315.039,Z 323.453,A -85,B 0,C 180,E1 -15626.102,E2 -15626.102} C_VEL
LIN {X 0,Y 314.865,Z 323.333,A -85,B 0,C 180,E1 -15630.518,E2 -15630.518} C_VEL
LIN {X 0,Y 314.886,Z 323.702,A -85,B 0,C 180,E1 -15632.458,E2 -15632.458} C_VEL
LIN {X 0,Y 315.91,Z 325.977,A -85,B 0,C 180,E1 -15632.858,E2 -15632.858} C_VEL
LIN {X 0,Y 317.992,Z 328.856,A -85,B 0,C 180,E1 -15633.54,E2 -15633.54} C_VEL
LIN {X 0,Y 322.346,Z 336.523,A -85,B 0,C 180,E1 -15635.083,E2 -15635.083} C_VEL
LIN {X 0,Y 326.419,Z 346.307,A -85,B 0,C 180,E1 -15636.814,E2 -15636.814} C_VEL
LIN {X 0,Y 327.672,Z 351.136,A -85,B 0,C 180,E1 -15637.591,E2 -15637.591} C_VEL
LIN {X 0,Y 325.549,Z 363.238,A -85,B 0,C 180,E1 -15638.967,E2 -15638.967} C_VEL
LIN {X 0,Y 323.688,Z 372.876,A -85,B 0,C 180,E1 -15640.334,E2 -15640.334} C_VEL
LIN {X 0,Y 321.761,Z 381.835,A -85,B 0,C 180,E1 -15641.865,E2 -15641.865} C_VEL
LIN {X 0,Y 319.664,Z 390.646,A -85,B 0,C 180,E1 -15643.721,E2 -15643.721} C_VEL
LIN {X 0,Y 317.899,Z 397.777,A -85,B 0,C 180,E1 -15645.599,E2 -15645.599} C_VEL
LIN {X 0,Y 316.519,Z 402.662,A -85,B 0,C 180,E1 -15647.171,E2 -15647.171} C_VEL
LIN {X 0,Y 315.105,Z 407.793,A -85,B 0,C 180,E1 -15649.291,E2 -15649.291} C_VEL
LIN {X 0,Y 314.092,Z 410.93,A -85,B 0,C 180,E1 -15650.989,E2 -15650.989} C_VEL
LIN {X 0,Y 313.501,Z 412.72,A -85,B 0,C 180,E1 -15652.27,E2 -15652.27} C_VEL
LIN {X 0,Y 313.003,Z 414.078,A -85,B 0,C 180,E1 -15653.554,E2 -15653.554} C_VEL
LIN {X 0,Y 312.541,Z 415.032,A -85,B 0,C 180,E1 -15654.84,E2 -15654.84} C_VEL
LIN {X 0,Y 312.102,Z 415.54,A -85,B 0,C 180,E1 -15656.126,E2 -15656.126} C_VEL
LIN {X 0,Y 311.773,Z 415.621,A -85,B 0,C 180,E1 -15657.416,E2 -15657.416} C_VEL
LIN {X 0,Y 311.587,Z 415.295,A -85,B 0,C 180,E1 -15658.708,E2 -15658.708} C_VEL
LIN {X 0,Y 311.504,Z 414.542,A -85,B 0,C 180,E1 -15660,E2 -15660} C_VEL
LIN {X 0,Y 311.484,Z 413.33,A -85,B 0,C 180,E1 -15661.293,E2 -15661.293} C_VEL
LIN {X 0,Y 311.615,Z 410.718,A -85,B 0,C 180,E1 -15663.232,E2 -15663.232} C_VEL
LIN {X 0,Y 311.856,Z 407.079,A -85,B 0,C 180,E1 -15665.172,E2 -15665.172} C_VEL
LIN {X 0,Y 312.095,Z 401.542,A -85,B 0,C 180,E1 -15667.4,E2 -15667.4} C_VEL
LIN {X 0,Y 312.544,Z 395.191,A -85,B 0,C 180,E1 -15669.383,E2 -15669.383} C_VEL
LIN {X 0,Y 313.23,Z 387.424,A -85,B 0,C 180,E1 -15671.322,E2 -15671.322} C_VEL
LIN {X 0,Y 314.009,Z 377.882,A -85,B 0,C 180,E1 -15673.263,E2 -15673.263} C_VEL
LIN {X 0,Y 314.986,Z 367.014,A -85,B 0,C 180,E1 -15675.033,E2 -15675.033} C_VEL
LIN {X 0,Y 315.868,Z 356.148,A -85,B 0,C 180,E1 -15676.48,E2 -15676.48} C_VEL
LIN {X 0,Y 316.655,Z 344.167,A -85,B 0,C 180,E1 -15677.766,E2 -15677.766} C_VEL
LIN {X 0,Y 317.237,Z 332.584,A -85,B 0,C 180,E1 -15678.765,E2 -15678.765} C_VEL
LIN {X 0,Y 314.32,Z 319.448,A -85,B 0,C 180,E1 -15679.777,E2 -15679.777} C_VEL
LIN {X 0,Y 312.066,Z 310.609,A -85,B 0,C 180,E1 -15680.352,E2 -15680.352} C_VEL
LIN {X 0,Y 312.332,Z 310.582,A -85,B 0,C 180,E1 -15683.893,E2 -15683.893} C_VEL
LIN {X 0,Y 312.489,Z 310.551,A -85,B 0,C 180,E1 -15686.732,E2 -15686.732} C_VEL
LIN {X 0,Y 312.535,Z 310.553,A -85,B 0,C 180,E1 -15689.651,E2 -15689.651} C_VEL
LIN {X 0,Y 312.522,Z 310.557,A -85,B 0,C 180,E1 -15693.689,E2 -15693.689} C_VEL
LIN {X 0,Y 312.539,Z 310.557,A -85,B 0,C 180,E1 -15697.383,E2 -15697.383} C_VEL
LIN {X 0,Y 312.492,Z 310.563,A -85,B 0,C 180,E1 -15700.709,E2 -15700.709} C_VEL
LIN {X 0,Y 312.454,Z 310.564,A -85,B 0,C 180,E1 -15704.21,E2 -15704.21} C_VEL
LIN {X 0,Y 312.486,Z 310.562,A -85,B 0,C 180,E1 -15707.919,E2 -15707.919} C_VEL
LIN {X 0,Y 312.498,Z 310.56,A -85,B 0,C 180,E1 -15710.971,E2 -15710.971} C_VEL
LIN {X 0,Y 312.533,Z 310.708,A -85,B 0,C 180,E1 -15714.051,E2 -15714.051} C_VEL
LIN {X 0,Y 312.831,Z 313.8,A -85,B 0,C 180,E1 -15716.226,E2 -15716.226} C_VEL
LIN {X 0,Y 312.497,Z 319.932,A -85,B 0,C 180,E1 -15720.345,E2 -15720.345} C_VEL
LIN {X 0,Y 312.371,Z 325.826,A -85,B 0,C 180,E1 -15724.153,E2 -15724.153} C_VEL
LIN {X 0,Y 312.346,Z 330.002,A -85,B 0,C 180,E1 -15726.713,E2 -15726.713} C_VEL
LIN {X 0,Y 316.951,Z 345.315,A -85,B 0,C 180,E1 -15727.738,E2 -15727.738} C_VEL
LIN {X 0,Y 319.577,Z 356.553,A -85,B 0,C 180,E1 -15728.66,E2 -15728.66} C_VEL
LIN {X 0,Y 320.888,Z 363.821,A -85,B 0,C 180,E1 -15729.354,E2 -15729.354} C_VEL
LIN {X 0,Y 319.784,Z 375.177,A -85,B 0,C 180,E1 -15730.418,E2 -15730.418} C_VEL
LIN {X 0,Y 318.517,Z 385.872,A -85,B 0,C 180,E1 -15731.697,E2 -15731.697} C_VEL
LIN {X 0,Y 317.244,Z 396.212,A -85,B 0,C 180,E1 -15733.262,E2 -15733.262} C_VEL
LIN {X 0,Y 315.853,Z 404.77,A -85,B 0,C 180,E1 -15734.844,E2 -15734.844} C_VEL
LIN {X 0,Y 314.569,Z 413.082,A -85,B 0,C 180,E1 -15736.762,E2 -15736.762} C_VEL
LIN {X 0,Y 313.635,Z 418.74,A -85,B 0,C 180,E1 -15738.365,E2 -15738.365} C_VEL
LIN {X 0,Y 312.703,Z 424.239,A -85,B 0,C 180,E1 -15740.296,E2 -15740.296} C_VEL
LIN {X 0,Y 312.095,Z 428.546,A -85,B 0,C 180,E1 -15742.235,E2 -15742.235} C_VEL
LIN {X 0,Y 311.753,Z 430.814,A -85,B 0,C 180,E1 -15743.528,E2 -15743.528} C_VEL
LIN {X 0,Y 311.417,Z 432.667,A -85,B 0,C 180,E1 -15744.821,E2 -15744.821} C_VEL
LIN {X 0,Y 311.267,Z 434.073,A -85,B 0,C 180,E1 -15746.116,E2 -15746.116} C_VEL
LIN {X 0,Y 311.176,Z 435.059,A -85,B 0,C 180,E1 -15747.411,E2 -15747.411} C_VEL
LIN {X 0,Y 311.061,Z 435.901,A -85,B 0,C 180,E1 -15750,E2 -15750} C_VEL
LIN {X 0,Y 311.17,Z 435.123,A -85,B 0,C 180,E1 -15752.589,E2 -15752.589} C_VEL
LIN {X 0,Y 311.4,Z 432.808,A -85,B 0,C 180,E1 -15755.18,E2 -15755.18} C_VEL
LIN {X 0,Y 311.955,Z 429.112,A -85,B 0,C 180,E1 -15757.574,E2 -15757.574} C_VEL
LIN {X 0,Y 312.658,Z 424.502,A -85,B 0,C 180,E1 -15759.706,E2 -15759.706} C_VEL
LIN {X 0,Y 313.568,Z 419.065,A -85,B 0,C 180,E1 -15761.637,E2 -15761.637} C_VEL
LIN {X 0,Y 314.694,Z 412.252,A -85,B 0,C 180,E1 -15763.562,E2 -15763.562} C_VEL
LIN {X 0,Y 316.052,Z 403.712,A -85,B 0,C 180,E1 -15765.477,E2 -15765.477} C_VEL
LIN {X 0,Y 317.484,Z 394.95,A -85,B 0,C 180,E1 -15767.056,E2 -15767.056} C_VEL
LIN {X 0,Y 318.535,Z 385.788,A -85,B 0,C 180,E1 -15768.425,E2 -15768.425} C_VEL
LIN {X 0,Y 319.846,Z 374.656,A -85,B 0,C 180,E1 -15769.745,E2 -15769.745} C_VEL
LIN {X 0,Y 320.949,Z 364.82,A -85,B 0,C 180,E1 -15770.664,E2 -15770.664} C_VEL
LIN {X 0,Y 319.703,Z 357.112,A -85,B 0,C 180,E1 -15771.397,E2 -15771.397} C_VEL
LIN {X 0,Y 316.797,Z 344.648,A -85,B 0,C 180,E1 -15772.419,E2 -15772.419} C_VEL
LIN {X 0,Y 312.883,Z 332,A -85,B 0,C 180,E1 -15773.263,E2 -15773.263} C_VEL
LIN {X 0,Y 312.353,Z 330.053,A -85,B 0,C 180,E1 -15773.377,E2 -15773.377} C_VEL
LIN {X 0,Y 312.406,Z 323.469,A -85,B 0,C 180,E1 -15777.463,E2 -15777.463} C_VEL
LIN {X 0,Y 312.592,Z 317.639,A -85,B 0,C 180,E1 -15781.311,E2 -15781.311} C_VEL
LIN {X 0,Y 312.858,Z 313.392,A -85,B 0,C 180,E1 -15784.166,E2 -15784.166} C_VEL
LIN {X 0,Y 312.514,Z 310.56,A -85,B 0,C 180,E1 -15786.312,E2 -15786.312} C_VEL
LIN {X 0,Y 312.506,Z 310.559,A -85,B 0,C 180,E1 -15790.125,E2 -15790.125} C_VEL
LIN {X 0,Y 312.46,Z 310.566,A -85,B 0,C 180,E1 -15793.965,E2 -15793.965} C_VEL
LIN {X 0,Y 312.486,Z 310.561,A -85,B 0,C 180,E1 -15797.919,E2 -15797.919} C_VEL
LIN {X 0,Y 312.496,Z 310.559,A -85,B 0,C 180,E1 -15800.971,E2 -15800.971} C_VEL
LIN {X 0,Y 312.452,Z 310.564,A -85,B 0,C 180,E1 -15804.209,E2 -15804.209} C_VEL
LIN {X 0,Y 312.321,Z 310.651,A -85,B 0,C 180,E1 -15806.831,E2 -15806.831} C_VEL
LIN {X 0,Y 311.942,Z 317.626,A -85,B 0,C 180,E1 -15811.482,E2 -15811.482} C_VEL
LIN {X 0,Y 311.816,Z 322.424,A -85,B 0,C 180,E1 -15814.706,E2 -15814.706} C_VEL
LIN {X 0,Y 311.098,Z 323.571,A -85,B 0,C 180,E1 -15815.393,E2 -15815.393} C_VEL
LIN {X 0,Y 308.21,Z 325.556,A -85,B 0,C 180,E1 -15816.457,E2 -15816.457} C_VEL
LIN {X 0,Y 305.328,Z 327.531,A -85,B 0,C 180,E1 -15817.54,E2 -15817.54} C_VEL
LIN {X 0,Y 304.645,Z 328.673,A -85,B 0,C 180,E1 -15818.248,E2 -15818.248} C_VEL
LIN {X 0,Y 304.642,Z 330.419,A -85,B 0,C 180,E1 -15819.402,E2 -15819.402} C_VEL
LIN {X 0,Y 307.447,Z 345.887,A -85,B 0,C 180,E1 -15820.367,E2 -15820.367} C_VEL
LIN {X 0,Y 309.693,Z 358.151,A -85,B 0,C 180,E1 -15821.357,E2 -15821.357} C_VEL
LIN {X 0,Y 308.995,Z 370.083,A -85,B 0,C 180,E1 -15822.46,E2 -15822.46} C_VEL
LIN {X 0,Y 308.106,Z 382.304,A -85,B 0,C 180,E1 -15823.874,E2 -15823.874} C_VEL
LIN {X 0,Y 307.017,Z 394.086,A -85,B 0,C 180,E1 -15825.585,E2 -15825.585} C_VEL
LIN {X 0,Y 306.064,Z 404.161,A -85,B 0,C 180,E1 -15827.4,E2 -15827.4} C_VEL
LIN {X 0,Y 305.306,Z 413.076,A -85,B 0,C 180,E1 -15829.388,E2 -15829.388} C_VEL
LIN {X 0,Y 304.715,Z 420.235,A -85,B 0,C 180,E1 -15831.378,E2 -15831.378} C_VEL
LIN {X 0,Y 304.281,Z 425.982,A -85,B 0,C 180,E1 -15833.368,E2 -15833.368} C_VEL
LIN {X 0,Y 304.154,Z 430.498,A -85,B 0,C 180,E1 -15835.361,E2 -15835.361} C_VEL
LIN {X 0,Y 303.95,Z 433.889,A -85,B 0,C 180,E1 -15837.349,E2 -15837.349} C_VEL
LIN {X 0,Y 303.923,Z 435.567,A -85,B 0,C 180,E1 -15838.675,E2 -15838.675} C_VEL
LIN {X 0,Y 303.988,Z 436.78,A -85,B 0,C 180,E1 -15840,E2 -15840} C_VEL
LIN {X 0,Y 304.094,Z 437.582,A -85,B 0,C 180,E1 -15841.324,E2 -15841.324} C_VEL
LIN {X 0,Y 304.292,Z 437.935,A -85,B 0,C 180,E1 -15842.648,E2 -15842.648} C_VEL
LIN {X 0,Y 304.564,Z 437.843,A -85,B 0,C 180,E1 -15843.97,E2 -15843.97} C_VEL
LIN {X 0,Y 304.878,Z 437.353,A -85,B 0,C 180,E1 -15845.291,E2 -15845.291} C_VEL
LIN {X 0,Y 305.049,Z 436.443,A -85,B 0,C 180,E1 -15846.615,E2 -15846.615} C_VEL
LIN {X 0,Y 305.396,Z 435.078,A -85,B 0,C 180,E1 -15847.937,E2 -15847.937} C_VEL
LIN {X 0,Y 306.52,Z 432.178,A -85,B 0,C 180,E1 -15849.902,E2 -15849.902} C_VEL
LIN {X 0,Y 307.605,Z 428.239,A -85,B 0,C 180,E1 -15851.866,E2 -15851.866} C_VEL
LIN {X 0,Y 308.973,Z 423.142,A -85,B 0,C 180,E1 -15853.818,E2 -15853.818} C_VEL
LIN {X 0,Y 310.693,Z 416.763,A -85,B 0,C 180,E1 -15855.75,E2 -15855.75} C_VEL
LIN {X 0,Y 312.647,Z 408.823,A -85,B 0,C 180,E1 -15857.666,E2 -15857.666} C_VEL
LIN {X 0,Y 315.086,Z 399.069,A -85,B 0,C 180,E1 -15859.547,E2 -15859.547} C_VEL
LIN {X 0,Y 317.109,Z 389.517,A -85,B 0,C 180,E1 -15861.057,E2 -15861.057} C_VEL
LIN {X 0,Y 319.323,Z 378.515,A -85,B 0,C 180,E1 -15862.465,E2 -15862.465} C_VEL
LIN {X 0,Y 320.376,Z 372.827,A -85,B 0,C 180,E1 -15863.086,E2 -15863.086} C_VEL
LIN {X 0,Y 318.858,Z 364.38,A -85,B 0,C 180,E1 -15864.353,E2 -15864.353} C_VEL
LIN {X 0,Y 315.585,Z 353.902,A -85,B 0,C 180,E1 -15866.053,E2 -15866.053} C_VEL
LIN {X 0,Y 312.607,Z 346.696,A -85,B 0,C 180,E1 -15867.324,E2 -15867.324} C_VEL
LIN {X 0,Y 310.276,Z 342.029,A -85,B 0,C 180,E1 -15868.224,E2 -15868.224} C_VEL
LIN {X 0,Y 308.869,Z 338.65,A -85,B 0,C 180,E1 -15868.869,E2 -15868.869} C_VEL
LIN {X 0,Y 309.973,Z 333.879,A -85,B 0,C 180,E1 -15872.976,E2 -15872.976} C_VEL
LIN {X 0,Y 310.268,Z 331.479,A -85,B 0,C 180,E1 -15875.368,E2 -15875.368} C_VEL
LIN {X 0,Y 310.24,Z 329.597,A -85,B 0,C 180,E1 -15877.708,E2 -15877.708} C_VEL
LIN {X 0,Y 310.126,Z 327.497,A -85,B 0,C 180,E1 -15881.086,E2 -15881.086} C_VEL
LIN {X 0,Y 309.823,Z 326.757,A -85,B 0,C 180,E1 -15883.457,E2 -15883.457} C_VEL
LIN {X 0,Y 309.11,Z 326.928,A -85,B 0,C 180,E1 -15886.682,E2 -15886.682} C_VEL
LIN {X 0,Y 308.732,Z 328.496,A -85,B 0,C 180,E1 -15890.084,E2 -15890.084} C_VEL
LIN {X 0,Y 309.372,Z 332.351,A -85,B 0,C 180,E1 -15892.167,E2 -15892.167} C_VEL
LIN {X 0,Y 308.921,Z 336.858,A -85,B 0,C 180,E1 -15894.467,E2 -15894.467} C_VEL
LIN {X 0,Y 307.735,Z 344.617,A -85,B 0,C 180,E1 -15898.313,E2 -15898.313} C_VEL
LIN {X 0,Y 307.105,Z 349.121,A -85,B 0,C 180,E1 -15900.415,E2 -15900.415} C_VEL
LIN {X 0,Y 307.224,Z 352.845,A -85,B 0,C 180,E1 -15901.377,E2 -15901.377} C_VEL
LIN {X 0,Y 308.81,Z 357.743,A -85,B 0,C 180,E1 -15902.088,E2 -15902.088} C_VEL
LIN {X 0,Y 310.061,Z 362.561,A -85,B 0,C 180,E1 -15902.689,E2 -15902.689} C_VEL
LIN {X 0,Y 312.547,Z 373.606,A -85,B 0,C 180,E1 -15903.992,E2 -15903.992} C_VEL
LIN {X 0,Y 314.426,Z 386.635,A -85,B 0,C 180,E1 -15905.487,E2 -15905.487} C_VEL
LIN {X 0,Y 314.625,Z 395.285,A -85,B 0,C 180,E1 -15906.446,E2 -15906.446} C_VEL
LIN {X 0,Y 314.166,Z 408.018,A -85,B 0,C 180,E1 -15907.994,E2 -15907.994} C_VEL
LIN {X 0,Y 313.831,Z 415.274,A -85,B 0,C 180,E1 -15909.004,E2 -15909.004} C_VEL
LIN {X 0,Y 311.535,Z 426.037,A -85,B 0,C 180,E1 -15910.564,E2 -15910.564} C_VEL
LIN {X 0,Y 309.676,Z 435.033,A -85,B 0,C 180,E1 -15912.159,E2 -15912.159} C_VEL
LIN {X 0,Y 307.886,Z 444.057,A -85,B 0,C 180,E1 -15914.102,E2 -15914.102} C_VEL
LIN {X 0,Y 306.185,Z 452.583,A -85,B 0,C 180,E1 -15916.392,E2 -15916.392} C_VEL
LIN {X 0,Y 305.008,Z 459.332,A -85,B 0,C 180,E1 -15918.705,E2 -15918.705} C_VEL
LIN {X 0,Y 304.334,Z 463.886,A -85,B 0,C 180,E1 -15920.697,E2 -15920.697} C_VEL
LIN {X 0,Y 303.922,Z 468.366,A -85,B 0,C 180,E1 -15923.36,E2 -15923.36} C_VEL
LIN {X 0,Y 303.791,Z 469.926,A -85,B 0,C 180,E1 -15924.69,E2 -15924.69} C_VEL
LIN {X 0,Y 303.809,Z 471.074,A -85,B 0,C 180,E1 -15926.021,E2 -15926.021} C_VEL
LIN {X 0,Y 303.772,Z 471.819,A -85,B 0,C 180,E1 -15927.348,E2 -15927.348} C_VEL
LIN {X 0,Y 303.901,Z 472.136,A -85,B 0,C 180,E1 -15928.675,E2 -15928.675} C_VEL
LIN {X 0,Y 304.094,Z 472.011,A -85,B 0,C 180,E1 -15930,E2 -15930} C_VEL
LIN {X 0,Y 303.798,Z 471.045,A -85,B 0,C 180,E1 -15932.652,E2 -15932.652} C_VEL
LIN {X 0,Y 303.842,Z 470.022,A -85,B 0,C 180,E1 -15933.979,E2 -15933.979} C_VEL
LIN {X 0,Y 303.933,Z 467.47,A -85,B 0,C 180,E1 -15936.113,E2 -15936.113} C_VEL
LIN {X 0,Y 304.061,Z 464.288,A -85,B 0,C 180,E1 -15937.972,E2 -15937.972} C_VEL
LIN {X 0,Y 304.466,Z 459.819,A -85,B 0,C 180,E1 -15939.969,E2 -15939.969} C_VEL
LIN {X 0,Y 305.674,Z 451.679,A -85,B 0,C 180,E1 -15942.954,E2 -15942.954} C_VEL
LIN {X 0,Y 307.159,Z 443.777,A -85,B 0,C 180,E1 -15945.256,E2 -15945.256} C_VEL
LIN {X 0,Y 308.756,Z 435.533,A -85,B 0,C 180,E1 -15947.212,E2 -15947.212} C_VEL
LIN {X 0,Y 310.86,Z 425.624,A -85,B 0,C 180,E1 -15949.137,E2 -15949.137} C_VEL
LIN {X 0,Y 313.438,Z 413.57,A -85,B 0,C 180,E1 -15951.024,E2 -15951.024} C_VEL
LIN {X 0,Y 314.157,Z 402.018,A -85,B 0,C 180,E1 -15952.667,E2 -15952.667} C_VEL
LIN {X 0,Y 314.481,Z 390.301,A -85,B 0,C 180,E1 -15954.124,E2 -15954.124} C_VEL
LIN {X 0,Y 313.429,Z 378.827,A -85,B 0,C 180,E1 -15955.542,E2 -15955.542} C_VEL
LIN {X 0,Y 311.115,Z 366.806,A -85,B 0,C 180,E1 -15957.076,E2 -15957.076} C_VEL
LIN {X 0,Y 308.243,Z 356.843,A -85,B 0,C 180,E1 -15958.462,E2 -15958.462} C_VEL
LIN {X 0,Y 307.198,Z 352.652,A -85,B 0,C 180,E1 -15959.028,E2 -15959.028} C_VEL
LIN {X 0,Y 308.644,Z 345.434,A -85,B 0,C 180,E1 -15963.127,E2 -15963.127} C_VEL
LIN {X 0,Y 310.16,Z 339.555,A -85,B 0,C 180,E1 -15966.83,E2 -15966.83} C_VEL
LIN {X 0,Y 310.342,Z 337.245,A -85,B 0,C 180,E1 -15968.518,E2 -15968.518} C_VEL
LIN {X 0,Y 309.797,Z 333.799,A -85,B 0,C 180,E1 -15971.528,E2 -15971.528} C_VEL
LIN {X 0,Y 309.266,Z 330.741,A -85,B 0,C 180,E1 -15974.787,E2 -15974.787} C_VEL
LIN {X 0,Y 308.754,Z 327.995,A -85,B 0,C 180,E1 -15978.691,E2 -15978.691} C_VEL
LIN {X 0,Y 308.436,Z 326.399,A -85,B 0,C 180,E1 -15982.032,E2 -15982.032} C_VEL
LIN {X 0,Y 308.194,Z 325.482,A -85,B 0,C 180,E1 -15985.243,E2 -15985.243} C_VEL
LIN {X 0,Y 308.03,Z 325.135,A -85,B 0,C 180,E1 -15988.347,E2 -15988.347} C_VEL
LIN {X 0,Y 308.003,Z 325.307,A -85,B 0,C 180,E1 -15991.02,E2 -15991.02} C_VEL
LIN {X 0,Y 309.033,Z 327.533,A -85,B 0,C 180,E1 -15991.472,E2 -15991.472} C_VEL
LIN {X 0,Y 310.499,Z 329.093,A -85,B 0,C 180,E1 -15991.976,E2 -15991.976} C_VEL
LIN {X 0,Y 315.176,Z 336.723,A -85,B 0,C 180,E1 -15993.771,E2 -15993.771} C_VEL
LIN {X 0,Y 318.596,Z 343.852,A -85,B 0,C 180,E1 -15995.221,E2 -15995.221} C_VEL
LIN {X 0,Y 321.402,Z 351.777,A -85,B 0,C 180,E1 -15996.694,E2 -15996.694} C_VEL
LIN {X 0,Y 321.777,Z 353.298,A -85,B 0,C 180,E1 -15996.956,E2 -15996.956} C_VEL
LIN {X 0,Y 319.536,Z 365.154,A -85,B 0,C 180,E1 -15998.383,E2 -15998.383} C_VEL
LIN {X 0,Y 317.327,Z 375.542,A -85,B 0,C 180,E1 -15999.923,E2 -15999.923} C_VEL
LIN {X 0,Y 314.933,Z 385.666,A -85,B 0,C 180,E1 -16001.795,E2 -16001.795} C_VEL
LIN {X 0,Y 312.788,Z 393.852,A -85,B 0,C 180,E1 -16003.688,E2 -16003.688} C_VEL
LIN {X 0,Y 310.93,Z 400.497,A -85,B 0,C 180,E1 -16005.603,E2 -16005.603} C_VEL
LIN {X 0,Y 309.352,Z 405.801,A -85,B 0,C 180,E1 -16007.537,E2 -16007.537} C_VEL
LIN {X 0,Y 307.962,Z 409.978,A -85,B 0,C 180,E1 -16009.481,E2 -16009.481} C_VEL
LIN {X 0,Y 307.201,Z 412.132,A -85,B 0,C 180,E1 -16010.785,E2 -16010.785} C_VEL
LIN {X 0,Y 306.558,Z 413.823,A -85,B 0,C 180,E1 -16012.094,E2 -16012.094} C_VEL
LIN {X 0,Y 306.024,Z 415.099,A -85,B 0,C 180,E1 -16013.406,E2 -16013.406} C_VEL
LIN {X 0,Y 305.537,Z 415.957,A -85,B 0,C 180,E1 -16014.721,E2 -16014.721} C_VEL
LIN {X 0,Y 305.083,Z 416.378,A -85,B 0,C 180,E1 -16016.037,E2 -16016.037} C_VEL
LIN {X 0,Y 304.741,Z 416.389,A -85,B 0,C 180,E1 -16017.356,E2 -16017.356} C_VEL
LIN {X 0,Y 304.547,Z 415.984,A -85,B 0,C 180,E1 -16018.678,E2 -16018.678} C_VEL
LIN {X 0,Y 304.43,Z 415.119,A -85,B 0,C 180,E1 -16020,E2 -16020} C_VEL
LIN {X 0,Y 304.415,Z 413.839,A -85,B 0,C 180,E1 -16021.323,E2 -16021.323} C_VEL
LIN {X 0,Y 304.56,Z 411.097,A -85,B 0,C 180,E1 -16023.307,E2 -16023.307} C_VEL
LIN {X 0,Y 304.78,Z 407.321,A -85,B 0,C 180,E1 -16025.292,E2 -16025.292} C_VEL
LIN {X 0,Y 305.01,Z 401.993,A -85,B 0,C 180,E1 -16027.437,E2 -16027.437} C_VEL
LIN {X 0,Y 305.529,Z 395.071,A -85,B 0,C 180,E1 -16029.6,E2 -16029.6} C_VEL
LIN {X 0,Y 306.227,Z 387.16,A -85,B 0,C 180,E1 -16031.585,E2 -16031.585} C_VEL
LIN {X 0,Y 306.886,Z 379.171,A -85,B 0,C 180,E1 -16033.239,E2 -16033.239} C_VEL
LIN {X 0,Y 307.855,Z 368.449,A -85,B 0,C 180,E1 -16035.051,E2 -16035.051} C_VEL
LIN {X 0,Y 308.783,Z 357.724,A -85,B 0,C 180,E1 -16036.529,E2 -16036.529} C_VEL
LIN {X 0,Y 309.61,Z 346.001,A -85,B 0,C 180,E1 -16037.844,E2 -16037.844} C_VEL
LIN {X 0,Y 310.366,Z 334.46,A -85,B 0,C 180,E1 -16038.879,E2 -16038.879} C_VEL
LIN {X 0,Y 307.808,Z 322.509,A -85,B 0,C 180,E1 -16039.858,E2 -16039.858} C_VEL
LIN {X 0,Y 305.05,Z 311.48,A -85,B 0,C 180,E1 -16040.631,E2 -16040.631} C_VEL
LIN {X 0,Y 305.338,Z 311.453,A -85,B 0,C 180,E1 -16044.476,E2 -16044.476} C_VEL
LIN {X 0,Y 305.464,Z 311.43,A -85,B 0,C 180,E1 -16047.397,E2 -16047.397} C_VEL
LIN {X 0,Y 305.458,Z 311.431,A -85,B 0,C 180,E1 -16050.41,E2 -16050.41} C_VEL
LIN {X 0,Y 305.467,Z 311.436,A -85,B 0,C 180,E1 -16054.078,E2 -16054.078} C_VEL
LIN {X 0,Y 305.498,Z 311.435,A -85,B 0,C 180,E1 -16056.737,E2 -16056.737} C_VEL
LIN {X 0,Y 305.457,Z 311.44,A -85,B 0,C 180,E1 -16060.6,E2 -16060.6} C_VEL
LIN {X 0,Y 305.428,Z 311.444,A -85,B 0,C 180,E1 -16063.655,E2 -16063.655} C_VEL
LIN {X 0,Y 305.457,Z 311.436,A -85,B 0,C 180,E1 -16067.414,E2 -16067.414} C_VEL
LIN {X 0,Y 305.46,Z 311.437,A -85,B 0,C 180,E1 -16069.892,E2 -16069.892} C_VEL
LIN {X 0,Y 305.481,Z 311.517,A -85,B 0,C 180,E1 -16073.632,E2 -16073.632} C_VEL
LIN {X 0,Y 305.89,Z 314.539,A -85,B 0,C 180,E1 -16075.804,E2 -16075.804} C_VEL
LIN {X 0,Y 305.533,Z 321.276,A -85,B 0,C 180,E1 -16080.359,E2 -16080.359} C_VEL
LIN {X 0,Y 305.39,Z 327.01,A -85,B 0,C 180,E1 -16084.071,E2 -16084.071} C_VEL
LIN {X 0,Y 305.338,Z 330.394,A -85,B 0,C 180,E1 -16086.164,E2 -16086.164} C_VEL
LIN {X 0,Y 309.617,Z 344.094,A -85,B 0,C 180,E1 -16087.096,E2 -16087.096} C_VEL
LIN {X 0,Y 312.509,Z 355.923,A -85,B 0,C 180,E1 -16088.075,E2 -16088.075} C_VEL
LIN {X 0,Y 314.189,Z 365.726,A -85,B 0,C 180,E1 -16089.029,E2 -16089.029} C_VEL
LIN {X 0,Y 312.944,Z 377.042,A -85,B 0,C 180,E1 -16090.143,E2 -16090.143} C_VEL
LIN {X 0,Y 311.708,Z 386.961,A -85,B 0,C 180,E1 -16091.384,E2 -16091.384} C_VEL
LIN {X 0,Y 310.478,Z 396.621,A -85,B 0,C 180,E1 -16092.886,E2 -16092.886} C_VEL
LIN {X 0,Y 309.016,Z 405.183,A -85,B 0,C 180,E1 -16094.5,E2 -16094.5} C_VEL
LIN {X 0,Y 307.68,Z 413.495,A -85,B 0,C 180,E1 -16096.46,E2 -16096.46} C_VEL
LIN {X 0,Y 306.685,Z 419.155,A -85,B 0,C 180,E1 -16098.098,E2 -16098.098} C_VEL
LIN {X 0,Y 305.731,Z 424.653,A -85,B 0,C 180,E1 -16100.072,E2 -16100.072} C_VEL
LIN {X 0,Y 305.03,Z 429.22,A -85,B 0,C 180,E1 -16102.197,E2 -16102.197} C_VEL
LIN {X 0,Y 304.372,Z 433.082,A -85,B 0,C 180,E1 -16104.701,E2 -16104.701} C_VEL
LIN {X 0,Y 304.191,Z 434.488,A -85,B 0,C 180,E1 -16106.026,E2 -16106.026} C_VEL
LIN {X 0,Y 304.092,Z 435.474,A -85,B 0,C 180,E1 -16107.351,E2 -16107.351} C_VEL
LIN {X 0,Y 303.974,Z 436.316,A -85,B 0,C 180,E1 -16110,E2 -16110} C_VEL
LIN {X 0,Y 304.085,Z 435.538,A -85,B 0,C 180,E1 -16112.649,E2 -16112.649} C_VEL
LIN {X 0,Y 304.356,Z 433.221,A -85,B 0,C 180,E1 -16115.3,E2 -16115.3} C_VEL
LIN {X 0,Y 304.908,Z 429.735,A -85,B 0,C 180,E1 -16117.634,E2 -16117.634} C_VEL
LIN {X 0,Y 305.676,Z 424.914,A -85,B 0,C 180,E1 -16119.93,E2 -16119.93} C_VEL
LIN {X 0,Y 306.63,Z 419.476,A -85,B 0,C 180,E1 -16121.905,E2 -16121.905} C_VEL
LIN {X 0,Y 307.801,Z 412.661,A -85,B 0,C 180,E1 -16123.872,E2 -16123.872} C_VEL
LIN {X 0,Y 309.246,Z 404.117,A -85,B 0,C 180,E1 -16125.826,E2 -16125.826} C_VEL
LIN {X 0,Y 310.727,Z 395.352,A -85,B 0,C 180,E1 -16127.439,E2 -16127.439} C_VEL
LIN {X 0,Y 311.979,Z 384.989,A -85,B 0,C 180,E1 -16128.997,E2 -16128.997} C_VEL
LIN {X 0,Y 313.41,Z 373.518,A -85,B 0,C 180,E1 -16130.339,E2 -16130.339} C_VEL
LIN {X 0,Y 314.245,Z 365.354,A -85,B 0,C 180,E1 -16131.113,E2 -16131.113} C_VEL
LIN {X 0,Y 311.886,Z 353.1,A -85,B 0,C 180,E1 -16132.286,E2 -16132.286} C_VEL
LIN {X 0,Y 308.725,Z 340.964,A -85,B 0,C 180,E1 -16133.252,E2 -16133.252} C_VEL
LIN {X 0,Y 305.336,Z 330.407,A -85,B 0,C 180,E1 -16133.961,E2 -16133.961} C_VEL
LIN {X 0,Y 305.429,Z 324.892,A -85,B 0,C 180,E1 -16137.401,E2 -16137.401} C_VEL
LIN {X 0,Y 305.579,Z 320.356,A -85,B 0,C 180,E1 -16140.396,E2 -16140.396} C_VEL
LIN {X 0,Y 305.902,Z 314.768,A -85,B 0,C 180,E1 -16144.199,E2 -16144.199} C_VEL
LIN {X 0,Y 305.491,Z 311.434,A -85,B 0,C 180,E1 -16146.555,E2 -16146.555} C_VEL
LIN {X 0,Y 305.457,Z 311.439,A -85,B 0,C 180,E1 -16150.6,E2 -16150.6} C_VEL
LIN {X 0,Y 305.428,Z 311.442,A -85,B 0,C 180,E1 -16153.655,E2 -16153.655} C_VEL
LIN {X 0,Y 305.457,Z 311.439,A -85,B 0,C 180,E1 -16157.414,E2 -16157.414} C_VEL
LIN {X 0,Y 305.46,Z 311.437,A -85,B 0,C 180,E1 -16159.892,E2 -16159.892} C_VEL
LIN {X 0,Y 305.419,Z 311.442,A -85,B 0,C 180,E1 -16163.648,E2 -16163.648} C_VEL
LIN {X 0,Y 305.29,Z 311.616,A -85,B 0,C 180,E1 -16166.856,E2 -16166.856} C_VEL
LIN {X 0,Y 304.903,Z 318.028,A -85,B 0,C 180,E1 -16171.152,E2 -16171.152} C_VEL
LIN {X 0,Y 304.77,Z 323.418,A -85,B 0,C 180,E1 -16174.772,E2 -16174.772} C_VEL
LIN {X 0,Y 304.645,Z 328.673,A -85,B 0,C 180,E1 -16178.248,E2 -16178.248} C_VEL
LIN {X 0,Y 304.541,Z 330.166,A -85,B 0,C 180,E1 -16178.765,E2 -16178.765} C_VEL
LIN {X 0,Y 304.183,Z 333.394,A -85,B 0,C 180,E1 -16179.283,E2 -16179.283} C_VEL
LIN {X 0,Y 303.509,Z 338.493,A -85,B 0,C 180,E1 -16179.724,E2 -16179.724} C_VEL
LIN {X 0,Y 301.952,Z 351.66,A -85,B 0,C 180,E1 -16180.555,E2 -16180.555} C_VEL
LIN {X 0,Y 302.264,Z 356.585,A -85,B 0,C 180,E1 -16180.958,E2 -16180.958} C_VEL
LIN {X 0,Y 302.719,Z 359.38,A -85,B 0,C 180,E1 -16181.208,E2 -16181.208} C_VEL
LIN {X 0,Y 301.889,Z 371.577,A -85,B 0,C 180,E1 -16182.384,E2 -16182.384} C_VEL
LIN {X 0,Y 301.055,Z 382.809,A -85,B 0,C 180,E1 -16183.732,E2 -16183.732} C_VEL
LIN {X 0,Y 299.995,Z 394.107,A -85,B 0,C 180,E1 -16185.413,E2 -16185.413} C_VEL
LIN {X 0,Y 299.088,Z 403.423,A -85,B 0,C 180,E1 -16187.101,E2 -16187.101} C_VEL
LIN {X 0,Y 298.277,Z 412.518,A -85,B 0,C 180,E1 -16189.135,E2 -16189.135} C_VEL
LIN {X 0,Y 297.671,Z 419.931,A -85,B 0,C 180,E1 -16191.172,E2 -16191.172} C_VEL
LIN {X 0,Y 297.215,Z 426.036,A -85,B 0,C 180,E1 -16193.287,E2 -16193.287} C_VEL
LIN {X 0,Y 297.07,Z 430.503,A -85,B 0,C 180,E1 -16195.25,E2 -16195.25} C_VEL
LIN {X 0,Y 296.868,Z 434.015,A -85,B 0,C 180,E1 -16197.286,E2 -16197.286} C_VEL
LIN {X 0,Y 296.828,Z 435.794,A -85,B 0,C 180,E1 -16198.643,E2 -16198.643} C_VEL
LIN {X 0,Y 296.895,Z 437.089,A -85,B 0,C 180,E1 -16200,E2 -16200} C_VEL
LIN {X 0,Y 297.007,Z 437.96,A -85,B 0,C 180,E1 -16201.356,E2 -16201.356} C_VEL
LIN {X 0,Y 297.231,Z 438.424,A -85,B 0,C 180,E1 -16202.71,E2 -16202.71} C_VEL
LIN {X 0,Y 297.516,Z 438.416,A -85,B 0,C 180,E1 -16204.064,E2 -16204.064} C_VEL
LIN {X 0,Y 297.837,Z 437.993,A -85,B 0,C 180,E1 -16205.416,E2 -16205.416} C_VEL
LIN {X 0,Y 298.027,Z 437.199,A -85,B 0,C 180,E1 -16206.771,E2 -16206.771} C_VEL
LIN {X 0,Y 298.428,Z 435.937,A -85,B 0,C 180,E1 -16208.123,E2 -16208.123} C_VEL
LIN {X 0,Y 299.601,Z 433.171,A -85,B 0,C 180,E1 -16210.133,E2 -16210.133} C_VEL
LIN {X 0,Y 300.773,Z 429.395,A -85,B 0,C 180,E1 -16212.14,E2 -16212.14} C_VEL
LIN {X 0,Y 302.212,Z 424.504,A -85,B 0,C 180,E1 -16214.133,E2 -16214.133} C_VEL
LIN {X 0,Y 304.037,Z 418.314,A -85,B 0,C 180,E1 -16216.104,E2 -16216.104} C_VEL
LIN {X 0,Y 306.107,Z 410.733,A -85,B 0,C 180,E1 -16218.056,E2 -16218.056} C_VEL
LIN {X 0,Y 308.669,Z 401.308,A -85,B 0,C 180,E1 -16219.97,E2 -16219.97} C_VEL
LIN {X 0,Y 311.22,Z 390.409,A -85,B 0,C 180,E1 -16221.769,E2 -16221.769} C_VEL
LIN {X 0,Y 313.721,Z 378.906,A -85,B 0,C 180,E1 -16223.274,E2 -16223.274} C_VEL
LIN {X 0,Y 314.504,Z 374.952,A -85,B 0,C 180,E1 -16223.718,E2 -16223.718} C_VEL
LIN {X 0,Y 313.231,Z 367.383,A -85,B 0,C 180,E1 -16224.958,E2 -16224.958} C_VEL
LIN {X 0,Y 310.501,Z 357.874,A -85,B 0,C 180,E1 -16226.61,E2 -16226.61} C_VEL
LIN {X 0,Y 306.239,Z 347.419,A -85,B 0,C 180,E1 -16228.635,E2 -16228.635} C_VEL
LIN {X 0,Y 304.019,Z 342.897,A -85,B 0,C 180,E1 -16229.613,E2 -16229.613} C_VEL
LIN {X 0,Y 302.593,Z 339.56,A -85,B 0,C 180,E1 -16230.343,E2 -16230.343} C_VEL
LIN {X 0,Y 303.53,Z 335.905,A -85,B 0,C 180,E1 -16233.759,E2 -16233.759} C_VEL
LIN {X 0,Y 303.82,Z 333.978,A -85,B 0,C 180,E1 -16235.941,E2 -16235.941} C_VEL
LIN {X 0,Y 303.8,Z 332.066,A -85,B 0,C 180,E1 -16238.654,E2 -16238.654} C_VEL
LIN {X 0,Y 303.838,Z 331.142,A -85,B 0,C 180,E1 -16240.366,E2 -16240.366} C_VEL
LIN {X 0,Y 303.747,Z 330.448,A -85,B 0,C 180,E1 -16242.234,E2 -16242.234} C_VEL
LIN {X 0,Y 303.458,Z 330.201,A -85,B 0,C 180,E1 -16244.114,E2 -16244.114} C_VEL
LIN {X 0,Y 303.126,Z 330.425,A -85,B 0,C 180,E1 -16245.95,E2 -16245.95} C_VEL
LIN {X 0,Y 302.726,Z 331.963,A -85,B 0,C 180,E1 -16249.455,E2 -16249.455} C_VEL
LIN {X 0,Y 302.579,Z 334.489,A -85,B 0,C 180,E1 -16252.159,E2 -16252.159} C_VEL
LIN {X 0,Y 302.182,Z 336.667,A -85,B 0,C 180,E1 -16253.625,E2 -16253.625} C_VEL
LIN {X 0,Y 301.302,Z 342.54,A -85,B 0,C 180,E1 -16256.493,E2 -16256.493} C_VEL
LIN {X 0,Y 301.023,Z 349.524,A -85,B 0,C 180,E1 -16259.094,E2 -16259.094} C_VEL
LIN {X 0,Y 301.289,Z 352.337,A -85,B 0,C 180,E1 -16259.953,E2 -16259.953} C_VEL
LIN {X 0,Y 304.19,Z 362.212,A -85,B 0,C 180,E1 -16261.466,E2 -16261.466} C_VEL
LIN {X 0,Y 306.564,Z 372.973,A -85,B 0,C 180,E1 -16262.868,E2 -16262.868} C_VEL
LIN {X 0,Y 308.248,Z 384.737,A -85,B 0,C 180,E1 -16264.329,E2 -16264.329} C_VEL
LIN {X 0,Y 308.782,Z 393.635,A -85,B 0,C 180,E1 -16265.425,E2 -16265.425} C_VEL
LIN {X 0,Y 308.112,Z 406.381,A -85,B 0,C 180,E1 -16267.004,E2 -16267.004} C_VEL
LIN {X 0,Y 307.356,Z 416.957,A -85,B 0,C 180,E1 -16268.54,E2 -16268.54} C_VEL
LIN {X 0,Y 304.95,Z 427.306,A -85,B 0,C 180,E1 -16270.127,E2 -16270.127} C_VEL
LIN {X 0,Y 302.63,Z 437.5,A -85,B 0,C 180,E1 -16272.079,E2 -16272.079} C_VEL
LIN {X 0,Y 300.799,Z 445.943,A -85,B 0,C 180,E1 -16274.066,E2 -16274.066} C_VEL
LIN {X 0,Y 299.295,Z 452.922,A -85,B 0,C 180,E1 -16276.073,E2 -16276.073} C_VEL
LIN {X 0,Y 298.023,Z 459.446,A -85,B 0,C 180,E1 -16278.437,E2 -16278.437} C_VEL
LIN {X 0,Y 297.301,Z 463.857,A -85,B 0,C 180,E1 -16280.475,E2 -16280.475} C_VEL
LIN {X 0,Y 297.022,Z 466.243,A -85,B 0,C 180,E1 -16281.838,E2 -16281.838} C_VEL
LIN {X 0,Y 296.739,Z 469.242,A -85,B 0,C 180,E1 -16284.119,E2 -16284.119} C_VEL
LIN {X 0,Y 296.717,Z 470.762,A -85,B 0,C 180,E1 -16285.925,E2 -16285.925} C_VEL
LIN {X 0,Y 296.692,Z 471.446,A -85,B 0,C 180,E1 -16287.285,E2 -16287.285} C_VEL
LIN {X 0,Y 297.034,Z 471.514,A -85,B 0,C 180,E1 -16290,E2 -16290} C_VEL
LIN {X 0,Y 296.876,Z 471.267,A -85,B 0,C 180,E1 -16291.357,E2 -16291.357} C_VEL
LIN {X 0,Y 296.751,Z 469.606,A -85,B 0,C 180,E1 -16294.074,E2 -16294.074} C_VEL
LIN {X 0,Y 296.842,Z 467.304,A -85,B 0,C 180,E1 -16296.072,E2 -16296.072} C_VEL
LIN {X 0,Y 296.995,Z 463.87,A -85,B 0,C 180,E1 -16298.163,E2 -16298.163} C_VEL
LIN {X 0,Y 297.44,Z 459.402,A -85,B 0,C 180,E1 -16300.207,E2 -16300.207} C_VEL
LIN {X 0,Y 298.524,Z 452.569,A -85,B 0,C 180,E1 -16302.924,E2 -16302.924} C_VEL
LIN {X 0,Y 300.083,Z 445.159,A -85,B 0,C 180,E1 -16305.277,E2 -16305.277} C_VEL
LIN {X 0,Y 301.758,Z 437.055,A -85,B 0,C 180,E1 -16307.36,E2 -16307.36} C_VEL
LIN {X 0,Y 303.857,Z 428.079,A -85,B 0,C 180,E1 -16309.244,E2 -16309.244} C_VEL
LIN {X 0,Y 306.537,Z 416.876,A -85,B 0,C 180,E1 -16311.168,E2 -16311.168} C_VEL
LIN {X 0,Y 307.769,Z 404.67,A -85,B 0,C 180,E1 -16313.032,E2 -16313.032} C_VEL
LIN {X 0,Y 308.396,Z 393.662,A -85,B 0,C 180,E1 -16314.514,E2 -16314.514} C_VEL
LIN {X 0,Y 307.921,Z 383.756,A -85,B 0,C 180,E1 -16315.826,E2 -16315.826} C_VEL
LIN {X 0,Y 306.048,Z 371.329,A -85,B 0,C 180,E1 -16317.526,E2 -16317.526} C_VEL
LIN {X 0,Y 303.639,Z 361.438,A -85,B 0,C 180,E1 -16318.989,E2 -16318.989} C_VEL
LIN {X 0,Y 301.657,Z 355.103,A -85,B 0,C 180,E1 -16320.018,E2 -16320.018} C_VEL
LIN {X 0,Y 300.729,Z 351.16,A -85,B 0,C 180,E1 -16320.62,E2 -16320.62} C_VEL
LIN {X 0,Y 302.25,Z 344.409,A -85,B 0,C 180,E1 -16324.728,E2 -16324.728} C_VEL
LIN {X 0,Y 303.265,Z 340.915,A -85,B 0,C 180,E1 -16327.052,E2 -16327.052} C_VEL
LIN {X 0,Y 303.424,Z 338.734,A -85,B 0,C 180,E1 -16328.711,E2 -16328.711} C_VEL
LIN {X 0,Y 302.845,Z 335.089,A -85,B 0,C 180,E1 -16332.046,E2 -16332.046} C_VEL
LIN {X 0,Y 302.53,Z 333.121,A -85,B 0,C 180,E1 -16334.181,E2 -16334.181} C_VEL
LIN {X 0,Y 301.962,Z 330.236,A -85,B 0,C 180,E1 -16338.141,E2 -16338.141} C_VEL
LIN {X 0,Y 301.685,Z 328.73,A -85,B 0,C 180,E1 -16341.024,E2 -16341.024} C_VEL
LIN {X 0,Y 301.391,Z 327.506,A -85,B 0,C 180,E1 -16344.702,E2 -16344.702} C_VEL
LIN {X 0,Y 301.23,Z 327.049,A -85,B 0,C 180,E1 -16347.547,E2 -16347.547} C_VEL
LIN {X 0,Y 301.174,Z 327.109,A -85,B 0,C 180,E1 -16349.352,E2 -16349.352} C_VEL
LIN {X 0,Y 302.489,Z 329.587,A -85,B 0,C 180,E1 -16349.996,E2 -16349.996} C_VEL
LIN {X 0,Y 304.492,Z 331.773,A -85,B 0,C 180,E1 -16350.797,E2 -16350.797} C_VEL
LIN {X 0,Y 305.07,Z 333.034,A -85,B 0,C 180,E1 -16351.095,E2 -16351.095} C_VEL
LIN {X 0,Y 306.529,Z 334.764,A -85,B 0,C 180,E1 -16351.653,E2 -16351.653} C_VEL
LIN {X 0,Y 311.54,Z 343.684,A -85,B 0,C 180,E1 -16353.852,E2 -16353.852} C_VEL
LIN {X 0,Y 314.957,Z 352.417,A -85,B 0,C 180,E1 -16355.672,E2 -16355.672} C_VEL
LIN {X 0,Y 315.922,Z 356.193,A -85,B 0,C 180,E1 -16356.395,E2 -16356.395} C_VEL
LIN {X 0,Y 313.631,Z 367.278,A -85,B 0,C 180,E1 -16357.781,E2 -16357.781} C_VEL
LIN {X 0,Y 311.039,Z 378.199,A -85,B 0,C 180,E1 -16359.499,E2 -16359.499} C_VEL
LIN {X 0,Y 308.476,Z 387.936,A -85,B 0,C 180,E1 -16361.4,E2 -16361.4} C_VEL
LIN {X 0,Y 306.223,Z 395.815,A -85,B 0,C 180,E1 -16363.329,E2 -16363.329} C_VEL
LIN {X 0,Y 304.271,Z 402.222,A -85,B 0,C 180,E1 -16365.281,E2 -16365.281} C_VEL
LIN {X 0,Y 302.557,Z 407.471,A -85,B 0,C 180,E1 -16367.32,E2 -16367.32} C_VEL
LIN {X 0,Y 301.122,Z 411.287,A -85,B 0,C 180,E1 -16369.239,E2 -16369.239} C_VEL
LIN {X 0,Y 300.31,Z 413.332,A -85,B 0,C 180,E1 -16370.571,E2 -16370.571} C_VEL
LIN {X 0,Y 299.62,Z 414.955,A -85,B 0,C 180,E1 -16371.909,E2 -16371.909} C_VEL
LIN {X 0,Y 299.048,Z 416.138,A -85,B 0,C 180,E1 -16373.252,E2 -16373.252} C_VEL
LIN {X 0,Y 298.535,Z 416.87,A -85,B 0,C 180,E1 -16374.597,E2 -16374.597} C_VEL
LIN {X 0,Y 298.064,Z 417.209,A -85,B 0,C 180,E1 -16375.944,E2 -16375.944} C_VEL
LIN {X 0,Y 297.71,Z 417.15,A -85,B 0,C 180,E1 -16377.294,E2 -16377.294} C_VEL
LIN {X 0,Y 297.49,Z 416.629,A -85,B 0,C 180,E1 -16378.646,E2 -16378.646} C_VEL
LIN {X 0,Y 297.358,Z 415.684,A -85,B 0,C 180,E1 -16380,E2 -16380} C_VEL
LIN {X 0,Y 297.348,Z 414.328,A -85,B 0,C 180,E1 -16381.354,E2 -16381.354} C_VEL
LIN {X 0,Y 297.506,Z 411.457,A -85,B 0,C 180,E1 -16383.386,E2 -16383.386} C_VEL
LIN {X 0,Y 297.711,Z 407.553,A -85,B 0,C 180,E1 -16385.418,E2 -16385.418} C_VEL
LIN {X 0,Y 297.957,Z 401.898,A -85,B 0,C 180,E1 -16387.659,E2 -16387.659} C_VEL
LIN {X 0,Y 298.499,Z 394.913,A -85,B 0,C 180,E1 -16389.828,E2 -16389.828} C_VEL
LIN {X 0,Y 299.22,Z 386.804,A -85,B 0,C 180,E1 -16391.86,E2 -16391.86} C_VEL
LIN {X 0,Y 300.107,Z 376.735,A -85,B 0,C 180,E1 -16393.889,E2 -16393.889} C_VEL
LIN {X 0,Y 301.096,Z 366.514,A -85,B 0,C 180,E1 -16395.571,E2 -16395.571} C_VEL
LIN {X 0,Y 302.049,Z 354.979,A -85,B 0,C 180,E1 -16397.111,E2 -16397.111} C_VEL
LIN {X 0,Y 302.897,Z 342.804,A -85,B 0,C 180,E1 -16398.43,E2 -16398.43} C_VEL
LIN {X 0,Y 303.255,Z 334.723,A -85,B 0,C 180,E1 -16399.145,E2 -16399.145} C_VEL
LIN {X 0,Y 300.465,Z 322.147,A -85,B 0,C 180,E1 -16400.192,E2 -16400.192} C_VEL
LIN {X 0,Y 298.04,Z 312.351,A -85,B 0,C 180,E1 -16400.85,E2 -16400.85} C_VEL
LIN {X 0,Y 298.331,Z 312.319,A -85,B 0,C 180,E1 -16405.09,E2 -16405.09} C_VEL
LIN {X 0,Y 298.43,Z 312.308,A -85,B 0,C 180,E1 -16408.099,E2 -16408.099} C_VEL
LIN {X 0,Y 298.396,Z 312.309,A -85,B 0,C 180,E1 -16412.016,E2 -16412.016} C_VEL
LIN {X 0,Y 298.433,Z 312.308,A -85,B 0,C 180,E1 -16416.068,E2 -16416.068} C_VEL
LIN {X 0,Y 298.411,Z 312.314,A -85,B 0,C 180,E1 -16419.486,E2 -16419.486} C_VEL
LIN {X 0,Y 298.4,Z 312.318,A -85,B 0,C 180,E1 -16423.103,E2 -16423.103} C_VEL
LIN {X 0,Y 298.405,Z 312.312,A -85,B 0,C 180,E1 -16426.921,E2 -16426.921} C_VEL
LIN {X 0,Y 298.398,Z 312.317,A -85,B 0,C 180,E1 -16431.008,E2 -16431.008} C_VEL
LIN {X 0,Y 298.439,Z 312.382,A -85,B 0,C 180,E1 -16433.195,E2 -16433.195} C_VEL
LIN {X 0,Y 298.894,Z 315.704,A -85,B 0,C 180,E1 -16435.645,E2 -16435.645} C_VEL
LIN {X 0,Y 298.559,Z 322.675,A -85,B 0,C 180,E1 -16440.374,E2 -16440.374} C_VEL
LIN {X 0,Y 298.417,Z 328.577,A -85,B 0,C 180,E1 -16444.213,E2 -16444.213} C_VEL
LIN {X 0,Y 298.404,Z 330.959,A -85,B 0,C 180,E1 -16445.593,E2 -16445.593} C_VEL
LIN {X 0,Y 302.658,Z 344.264,A -85,B 0,C 180,E1 -16446.526,E2 -16446.526} C_VEL
LIN {X 0,Y 305.615,Z 356.184,A -85,B 0,C 180,E1 -16447.543,E2 -16447.543} C_VEL
LIN {X 0,Y 307.478,Z 366.13,A -85,B 0,C 180,E1 -16448.549,E2 -16448.549} C_VEL
LIN {X 0,Y 306.304,Z 377.445,A -85,B 0,C 180,E1 -16449.694,E2 -16449.694} C_VEL
LIN {X 0,Y 304.818,Z 388.806,A -85,B 0,C 180,E1 -16451.168,E2 -16451.168} C_VEL
LIN {X 0,Y 303.412,Z 398.914,A -85,B 0,C 180,E1 -16452.823,E2 -16452.823} C_VEL
LIN {X 0,Y 301.963,Z 407.115,A -85,B 0,C 180,E1 -16454.475,E2 -16454.475} C_VEL
LIN {X 0,Y 300.557,Z 415.11,A -85,B 0,C 180,E1 -16456.477,E2 -16456.477} C_VEL
LIN {X 0,Y 299.364,Z 421.536,A -85,B 0,C 180,E1 -16458.489,E2 -16458.489} C_VEL
LIN {X 0,Y 298.465,Z 426.64,A -85,B 0,C 180,E1 -16460.513,E2 -16460.513} C_VEL
LIN {X 0,Y 297.981,Z 429.853,A -85,B 0,C 180,E1 -16462.134,E2 -16462.134} C_VEL
LIN {X 0,Y 297.329,Z 433.496,A -85,B 0,C 180,E1 -16464.575,E2 -16464.575} C_VEL
LIN {X 0,Y 297.12,Z 434.904,A -85,B 0,C 180,E1 -16465.931,E2 -16465.931} C_VEL
LIN {X 0,Y 297.008,Z 435.889,A -85,B 0,C 180,E1 -16467.287,E2 -16467.287} C_VEL
LIN {X 0,Y 296.886,Z 436.731,A -85,B 0,C 180,E1 -16470,E2 -16470} C_VEL
LIN {X 0,Y 296.902,Z 436.538,A -85,B 0,C 180,E1 -16471.356,E2 -16471.356} C_VEL
LIN {X 0,Y 297.001,Z 435.953,A -85,B 0,C 180,E1 -16472.713,E2 -16472.713} C_VEL
LIN {X 0,Y 297.315,Z 433.634,A -85,B 0,C 180,E1 -16475.426,E2 -16475.426} C_VEL
LIN {X 0,Y 297.844,Z 430.401,A -85,B 0,C 180,E1 -16477.673,E2 -16477.673} C_VEL
LIN {X 0,Y 298.69,Z 425.326,A -85,B 0,C 180,E1 -16480.164,E2 -16480.164} C_VEL
LIN {X 0,Y 299.71,Z 419.886,A -85,B 0,C 180,E1 -16482.184,E2 -16482.184} C_VEL
LIN {X 0,Y 300.933,Z 413.069,A -85,B 0,C 180,E1 -16484.195,E2 -16484.195} C_VEL
LIN {X 0,Y 302.452,Z 404.523,A -85,B 0,C 180,E1 -16486.191,E2 -16486.191} C_VEL
LIN {X 0,Y 303.98,Z 395.772,A -85,B 0,C 180,E1 -16487.836,E2 -16487.836} C_VEL
LIN {X 0,Y 305.29,Z 385.387,A -85,B 0,C 180,E1 -16489.43,E2 -16489.43} C_VEL
LIN {X 0,Y 306.785,Z 373.909,A -85,B 0,C 180,E1 -16490.799,E2 -16490.799} C_VEL
LIN {X 0,Y 307.478,Z 365.91,A -85,B 0,C 180,E1 -16491.585,E2 -16491.585} C_VEL
LIN {X 0,Y 305.006,Z 353.378,A -85,B 0,C 180,E1 -16492.825,E2 -16492.825} C_VEL
LIN {X 0,Y 301.792,Z 341.169,A -85,B 0,C 180,E1 -16493.826,E2 -16493.826} C_VEL
LIN {X 0,Y 298.384,Z 330.775,A -85,B 0,C 180,E1 -16494.548,E2 -16494.548} C_VEL
LIN {X 0,Y 298.498,Z 324.161,A -85,B 0,C 180,E1 -16498.759,E2 -16498.759} C_VEL
LIN {X 0,Y 298.758,Z 318.256,A -85,B 0,C 180,E1 -16502.756,E2 -16502.756} C_VEL
LIN {X 0,Y 298.883,Z 315.595,A -85,B 0,C 180,E1 -16504.614,E2 -16504.614} C_VEL
LIN {X 0,Y 298.418,Z 312.316,A -85,B 0,C 180,E1 -16507.022,E2 -16507.022} C_VEL
LIN {X 0,Y 298.389,Z 312.32,A -85,B 0,C 180,E1 -16511.088,E2 -16511.088} C_VEL
LIN {X 0,Y 298.4,Z 312.319,A -85,B 0,C 180,E1 -16513.103,E2 -16513.103} C_VEL
LIN {X 0,Y 298.405,Z 312.317,A -85,B 0,C 180,E1 -16516.921,E2 -16516.921} C_VEL
LIN {X 0,Y 298.396,Z 312.314,A -85,B 0,C 180,E1 -16521.008,E2 -16521.008} C_VEL
LIN {X 0,Y 298.344,Z 312.323,A -85,B 0,C 180,E1 -16523.92,E2 -16523.92} C_VEL
LIN {X 0,Y 298.246,Z 312.445,A -85,B 0,C 180,E1 -16526.779,E2 -16526.779} C_VEL
LIN {X 0,Y 297.871,Z 318.386,A -85,B 0,C 180,E1 -16530.807,E2 -16530.807} C_VEL
LIN {X 0,Y 297.75,Z 322.73,A -85,B 0,C 180,E1 -16533.759,E2 -16533.759} C_VEL
LIN {X 0,Y 297.604,Z 328.826,A -85,B 0,C 180,E1 -16537.8,E2 -16537.8} C_VEL
LIN {X 0,Y 297.593,Z 330.912,A -85,B 0,C 180,E1 -16539.162,E2 -16539.162} C_VEL
LIN {X 0,Y 300.106,Z 344.63,A -85,B 0,C 180,E1 -16539.996,E2 -16539.996} C_VEL
LIN {X 0,Y 302.264,Z 356.585,A -85,B 0,C 180,E1 -16540.958,E2 -16540.958} C_VEL
LIN {X 0,Y 302.382,Z 360.186,A -85,B 0,C 180,E1 -16541.269,E2 -16541.269} C_VEL
LIN {X 0,Y 301.151,Z 365.471,A -85,B 0,C 180,E1 -16541.72,E2 -16541.72} C_VEL
LIN {X 0,Y 295.137,Z 378.723,A -85,B 0,C 180,E1 -16543.027,E2 -16543.027} C_VEL
LIN {X 0,Y 293.983,Z 383.617,A -85,B 0,C 180,E1 -16543.65,E2 -16543.65} C_VEL
LIN {X 0,Y 292.849,Z 395.072,A -85,B 0,C 180,E1 -16545.405,E2 -16545.405} C_VEL
LIN {X 0,Y 291.959,Z 404.298,A -85,B 0,C 180,E1 -16547.134,E2 -16547.134} C_VEL
LIN {X 0,Y 291.145,Z 413.343,A -85,B 0,C 180,E1 -16549.218,E2 -16549.218} C_VEL
LIN {X 0,Y 290.556,Z 420.685,A -85,B 0,C 180,E1 -16551.305,E2 -16551.305} C_VEL
LIN {X 0,Y 290.113,Z 426.373,A -85,B 0,C 180,E1 -16553.33,E2 -16553.33} C_VEL
LIN {X 0,Y 289.944,Z 431.809,A -85,B 0,C 180,E1 -16555.83,E2 -16555.83} C_VEL
LIN {X 0,Y 289.788,Z 434.112,A -85,B 0,C 180,E1 -16557.22,E2 -16557.22} C_VEL
LIN {X 0,Y 289.736,Z 435.965,A -85,B 0,C 180,E1 -16558.61,E2 -16558.61} C_VEL
LIN {X 0,Y 289.802,Z 437.392,A -85,B 0,C 180,E1 -16560,E2 -16560} C_VEL
LIN {X 0,Y 289.92,Z 438.338,A -85,B 0,C 180,E1 -16561.389,E2 -16561.389} C_VEL
LIN {X 0,Y 290.153,Z 438.868,A -85,B 0,C 180,E1 -16562.777,E2 -16562.777} C_VEL
LIN {X 0,Y 290.47,Z 438.991,A -85,B 0,C 180,E1 -16564.162,E2 -16564.162} C_VEL
LIN {X 0,Y 290.8,Z 438.651,A -85,B 0,C 180,E1 -16565.547,E2 -16565.547} C_VEL
LIN {X 0,Y 291.006,Z 437.927,A -85,B 0,C 180,E1 -16566.936,E2 -16566.936} C_VEL
LIN {X 0,Y 291.472,Z 436.782,A -85,B 0,C 180,E1 -16568.318,E2 -16568.318} C_VEL
LIN {X 0,Y 292.687,Z 434.198,A -85,B 0,C 180,E1 -16570.375,E2 -16570.375} C_VEL
LIN {X 0,Y 293.939,Z 430.603,A -85,B 0,C 180,E1 -16572.427,E2 -16572.427} C_VEL
LIN {X 0,Y 295.463,Z 425.877,A -85,B 0,C 180,E1 -16574.463,E2 -16574.463} C_VEL
LIN {X 0,Y 297.778,Z 418.846,A -85,B 0,C 180,E1 -16576.805,E2 -16576.805} C_VEL
LIN {X 0,Y 300.008,Z 411.232,A -85,B 0,C 180,E1 -16578.79,E2 -16578.79} C_VEL
LIN {X 0,Y 302.768,Z 401.94,A -85,B 0,C 180,E1 -16580.732,E2 -16580.732} C_VEL
LIN {X 0,Y 305.26,Z 391.957,A -85,B 0,C 180,E1 -16582.426,E2 -16582.426} C_VEL
LIN {X 0,Y 308.11,Z 380.095,A -85,B 0,C 180,E1 -16584.04,E2 -16584.04} C_VEL
LIN {X 0,Y 308.713,Z 377.071,A -85,B 0,C 180,E1 -16584.408,E2 -16584.408} C_VEL
LIN {X 0,Y 307.445,Z 369.462,A -85,B 0,C 180,E1 -16585.743,E2 -16585.743} C_VEL
LIN {X 0,Y 304.943,Z 360.437,A -85,B 0,C 180,E1 -16587.448,E2 -16587.448} C_VEL
LIN {X 0,Y 302.373,Z 353.61,A -85,B 0,C 180,E1 -16588.873,E2 -16588.873} C_VEL
LIN {X 0,Y 298.242,Z 344.447,A -85,B 0,C 180,E1 -16591.02,E2 -16591.02} C_VEL
LIN {X 0,Y 296.559,Z 340.83,A -85,B 0,C 180,E1 -16591.945,E2 -16591.945} C_VEL
LIN {X 0,Y 296.557,Z 340.318,A -85,B 0,C 180,E1 -16592.223,E2 -16592.223} C_VEL
LIN {X 0,Y 297.155,Z 338.094,A -85,B 0,C 180,E1 -16594.585,E2 -16594.585} C_VEL
LIN {X 0,Y 297.374,Z 336.583,A -85,B 0,C 180,E1 -16596.53,E2 -16596.53} C_VEL
LIN {X 0,Y 297.476,Z 334.8,A -85,B 0,C 180,E1 -16599.635,E2 -16599.635} C_VEL
LIN {X 0,Y 297.511,Z 334.096,A -85,B 0,C 180,E1 -16601.409,E2 -16601.409} C_VEL
LIN {X 0,Y 297.395,Z 333.764,A -85,B 0,C 180,E1 -16603.261,E2 -16603.261} C_VEL
LIN {X 0,Y 297.1,Z 333.909,A -85,B 0,C 180,E1 -16605.207,E2 -16605.207} C_VEL
LIN {X 0,Y 296.752,Z 335.226,A -85,B 0,C 180,E1 -16608.461,E2 -16608.461} C_VEL
LIN {X 0,Y 296.76,Z 336.494,A -85,B 0,C 180,E1 -16610.251,E2 -16610.251} C_VEL
LIN {X 0,Y 296.681,Z 338.325,A -85,B 0,C 180,E1 -16611.982,E2 -16611.982} C_VEL
LIN {X 0,Y 296.148,Z 341.213,A -85,B 0,C 180,E1 -16613.791,E2 -16613.791} C_VEL
LIN {X 0,Y 295.377,Z 346.676,A -85,B 0,C 180,E1 -16616.384,E2 -16616.384} C_VEL
LIN {X 0,Y 295.21,Z 351.594,A -85,B 0,C 180,E1 -16618.215,E2 -16618.215} C_VEL
LIN {X 0,Y 297.379,Z 358.043,A -85,B 0,C 180,E1 -16619.467,E2 -16619.467} C_VEL
LIN {X 0,Y 299.573,Z 366.396,A -85,B 0,C 180,E1 -16620.796,E2 -16620.796} C_VEL
LIN {X 0,Y 301.576,Z 377.242,A -85,B 0,C 180,E1 -16622.321,E2 -16622.321} C_VEL
LIN {X 0,Y 302.848,Z 390.113,A -85,B 0,C 180,E1 -16624.041,E2 -16624.041} C_VEL
LIN {X 0,Y 302.869,Z 397.073,A -85,B 0,C 180,E1 -16624.949,E2 -16624.949} C_VEL
LIN {X 0,Y 301.847,Z 409.917,A -85,B 0,C 180,E1 -16626.683,E2 -16626.683} C_VEL
LIN {X 0,Y 300.895,Z 418.762,A -85,B 0,C 180,E1 -16628.055,E2 -16628.055} C_VEL
LIN {X 0,Y 297.962,Z 430.363,A -85,B 0,C 180,E1 -16630.001,E2 -16630.001} C_VEL
LIN {X 0,Y 295.595,Z 439.87,A -85,B 0,C 180,E1 -16631.996,E2 -16631.996} C_VEL
LIN {X 0,Y 293.457,Z 448.939,A -85,B 0,C 180,E1 -16634.37,E2 -16634.37} C_VEL
LIN {X 0,Y 291.742,Z 456.162,A -85,B 0,C 180,E1 -16636.77,E2 -16636.77} C_VEL
LIN {X 0,Y 290.762,Z 461.128,A -85,B 0,C 180,E1 -16638.851,E2 -16638.851} C_VEL
LIN {X 0,Y 290.094,Z 465.043,A -85,B 0,C 180,E1 -16640.94,E2 -16640.94} C_VEL
LIN {X 0,Y 289.769,Z 467.98,A -85,B 0,C 180,E1 -16643.035,E2 -16643.035} C_VEL
LIN {X 0,Y 289.627,Z 470.454,A -85,B 0,C 180,E1 -16645.825,E2 -16645.825} C_VEL
LIN {X 0,Y 289.614,Z 471.036,A -85,B 0,C 180,E1 -16647.218,E2 -16647.218} C_VEL
LIN {X 0,Y 289.956,Z 471.088,A -85,B 0,C 180,E1 -16650,E2 -16650} C_VEL
LIN {X 0,Y 289.777,Z 470.851,A -85,B 0,C 180,E1 -16651.39,E2 -16651.39} C_VEL
LIN {X 0,Y 289.663,Z 469.189,A -85,B 0,C 180,E1 -16654.174,E2 -16654.174} C_VEL
LIN {X 0,Y 289.748,Z 467.145,A -85,B 0,C 180,E1 -16656.022,E2 -16656.022} C_VEL
LIN {X 0,Y 289.928,Z 463.452,A -85,B 0,C 180,E1 -16658.363,E2 -16658.363} C_VEL
LIN {X 0,Y 290.89,Z 455.964,A -85,B 0,C 180,E1 -16661.851,E2 -16661.851} C_VEL
LIN {X 0,Y 292.239,Z 449.646,A -85,B 0,C 180,E1 -16664.271,E2 -16664.271} C_VEL
LIN {X 0,Y 293.98,Z 441.737,A -85,B 0,C 180,E1 -16666.671,E2 -16666.671} C_VEL
LIN {X 0,Y 295.961,Z 433.535,A -85,B 0,C 180,E1 -16668.698,E2 -16668.698} C_VEL
LIN {X 0,Y 298.521,Z 423.7,A -85,B 0,C 180,E1 -16670.68,E2 -16670.68} C_VEL
LIN {X 0,Y 300.415,Z 416.067,A -85,B 0,C 180,E1 -16671.982,E2 -16671.982} C_VEL
LIN {X 0,Y 301.617,Z 404.799,A -85,B 0,C 180,E1 -16673.791,E2 -16673.791} C_VEL
LIN {X 0,Y 302.369,Z 394.342,A -85,B 0,C 180,E1 -16675.283,E2 -16675.283} C_VEL
LIN {X 0,Y 301.837,Z 382.923,A -85,B 0,C 180,E1 -16676.916,E2 -16676.916} C_VEL
LIN {X 0,Y 300.213,Z 371.909,A -85,B 0,C 180,E1 -16678.572,E2 -16678.572} C_VEL
LIN {X 0,Y 297.749,Z 361.142,A -85,B 0,C 180,E1 -16680.333,E2 -16680.333} C_VEL
LIN {X 0,Y 295.787,Z 354.767,A -85,B 0,C 180,E1 -16681.516,E2 -16681.516} C_VEL
LIN {X 0,Y 294.509,Z 350.517,A -85,B 0,C 180,E1 -16682.323,E2 -16682.323} C_VEL
LIN {X 0,Y 294.395,Z 349.497,A -85,B 0,C 180,E1 -16682.489,E2 -16682.489} C_VEL
LIN {X 0,Y 296,Z 343.516,A -85,B 0,C 180,E1 -16686.412,E2 -16686.412} C_VEL
LIN {X 0,Y 296.512,Z 341.283,A -85,B 0,C 180,E1 -16688.044,E2 -16688.044} C_VEL
LIN {X 0,Y 296.261,Z 338.343,A -85,B 0,C 180,E1 -16690.614,E2 -16690.614} C_VEL
LIN {X 0,Y 295.604,Z 334.728,A -85,B 0,C 180,E1 -16694.5,E2 -16694.5} C_VEL
LIN {X 0,Y 295.133,Z 332.123,A -85,B 0,C 180,E1 -16698.182,E2 -16698.182} C_VEL
LIN {X 0,Y 294.759,Z 330.299,A -85,B 0,C 180,E1 -16701.89,E2 -16701.89} C_VEL
LIN {X 0,Y 294.53,Z 329.335,A -85,B 0,C 180,E1 -16705.062,E2 -16705.062} C_VEL
LIN {X 0,Y 294.428,Z 329.092,A -85,B 0,C 180,E1 -16707.35,E2 -16707.35} C_VEL
LIN {X 0,Y 294.992,Z 330.478,A -85,B 0,C 180,E1 -16707.753,E2 -16707.753} C_VEL
LIN {X 0,Y 297.762,Z 333.463,A -85,B 0,C 180,E1 -16709.075,E2 -16709.075} C_VEL
LIN {X 0,Y 298.589,Z 335.024,A -85,B 0,C 180,E1 -16709.544,E2 -16709.544} C_VEL
LIN {X 0,Y 299.893,Z 336.522,A -85,B 0,C 180,E1 -16710.123,E2 -16710.123} C_VEL
LIN {X 0,Y 304.278,Z 343.595,A -85,B 0,C 180,E1 -16712.224,E2 -16712.224} C_VEL
LIN {X 0,Y 307.512,Z 350.361,A -85,B 0,C 180,E1 -16713.915,E2 -16713.915} C_VEL
LIN {X 0,Y 310.205,Z 358.803,A -85,B 0,C 180,E1 -16715.744,E2 -16715.744} C_VEL
LIN {X 0,Y 307.483,Z 370.484,A -85,B 0,C 180,E1 -16717.312,E2 -16717.312} C_VEL
LIN {X 0,Y 304.759,Z 380.968,A -85,B 0,C 180,E1 -16719.057,E2 -16719.057} C_VEL
LIN {X 0,Y 302.054,Z 390.24,A -85,B 0,C 180,E1 -16720.989,E2 -16720.989} C_VEL
LIN {X 0,Y 299.7,Z 397.832,A -85,B 0,C 180,E1 -16722.955,E2 -16722.955} C_VEL
LIN {X 0,Y 297.621,Z 403.949,A -85,B 0,C 180,E1 -16724.945,E2 -16724.945} C_VEL
LIN {X 0,Y 295.943,Z 408.536,A -85,B 0,C 180,E1 -16726.821,E2 -16726.821} C_VEL
LIN {X 0,Y 294.284,Z 412.625,A -85,B 0,C 180,E1 -16728.986,E2 -16728.986} C_VEL
LIN {X 0,Y 293.421,Z 414.571,A -85,B 0,C 180,E1 -16730.348,E2 -16730.348} C_VEL
LIN {X 0,Y 292.685,Z 416.081,A -85,B 0,C 180,E1 -16731.716,E2 -16731.716} C_VEL
LIN {X 0,Y 292.075,Z 417.133,A -85,B 0,C 180,E1 -16733.09,E2 -16733.09} C_VEL
LIN {X 0,Y 291.535,Z 417.791,A -85,B 0,C 180,E1 -16734.467,E2 -16734.467} C_VEL
LIN {X 0,Y 291.047,Z 418.055,A -85,B 0,C 180,E1 -16735.846,E2 -16735.846} C_VEL
LIN {X 0,Y 290.681,Z 417.871,A -85,B 0,C 180,E1 -16737.228,E2 -16737.228} C_VEL
LIN {X 0,Y 290.42,Z 417.256,A -85,B 0,C 180,E1 -16738.613,E2 -16738.613} C_VEL
LIN {X 0,Y 290.288,Z 416.238,A -85,B 0,C 180,E1 -16740,E2 -16740} C_VEL
LIN {X 0,Y 290.284,Z 414.792,A -85,B 0,C 180,E1 -16741.387,E2 -16741.387} C_VEL
LIN {X 0,Y 290.435,Z 411.774,A -85,B 0,C 180,E1 -16743.468,E2 -16743.468} C_VEL
LIN {X 0,Y 290.646,Z 407.706,A -85,B 0,C 180,E1 -16745.551,E2 -16745.551} C_VEL
LIN {X 0,Y 290.93,Z 401.639,A -85,B 0,C 180,E1 -16747.928,E2 -16747.928} C_VEL
LIN {X 0,Y 291.488,Z 394.743,A -85,B 0,C 180,E1 -16750.067,E2 -16750.067} C_VEL
LIN {X 0,Y 292.223,Z 386.371,A -85,B 0,C 180,E1 -16752.148,E2 -16752.148} C_VEL
LIN {X 0,Y 293.168,Z 376.064,A -85,B 0,C 180,E1 -16754.224,E2 -16754.224} C_VEL
LIN {X 0,Y 294.19,Z 365.47,A -85,B 0,C 180,E1 -16755.946,E2 -16755.946} C_VEL
LIN {X 0,Y 295.177,Z 353.209,A -85,B 0,C 180,E1 -16757.57,E2 -16757.57} C_VEL
LIN {X 0,Y 296.054,Z 340.804,A -85,B 0,C 180,E1 -16758.871,E2 -16758.871} C_VEL
LIN {X 0,Y 296.29,Z 335.97,A -85,B 0,C 180,E1 -16759.305,E2 -16759.305} C_VEL
LIN {X 0,Y 293.737,Z 324.326,A -85,B 0,C 180,E1 -16760.315,E2 -16760.315} C_VEL
LIN {X 0,Y 291.026,Z 313.267,A -85,B 0,C 180,E1 -16761.098,E2 -16761.098} C_VEL
LIN {X 0,Y 291.22,Z 313.211,A -85,B 0,C 180,E1 -16764.221,E2 -16764.221} C_VEL
LIN {X 0,Y 291.358,Z 313.185,A -85,B 0,C 180,E1 -16767.278,E2 -16767.278} C_VEL
LIN {X 0,Y 291.334,Z 313.189,A -85,B 0,C 180,E1 -16770.437,E2 -16770.437} C_VEL
LIN {X 0,Y 291.347,Z 313.195,A -85,B 0,C 180,E1 -16773.698,E2 -16773.698} C_VEL
LIN {X 0,Y 291.396,Z 313.191,A -85,B 0,C 180,E1 -16777.259,E2 -16777.259} C_VEL
LIN {X 0,Y 291.336,Z 313.199,A -85,B 0,C 180,E1 -16780.642,E2 -16780.642} C_VEL
LIN {X 0,Y 291.292,Z 313.199,A -85,B 0,C 180,E1 -16784.402,E2 -16784.402} C_VEL
LIN {X 0,Y 291.328,Z 313.195,A -85,B 0,C 180,E1 -16788.404,E2 -16788.404} C_VEL
LIN {X 0,Y 291.356,Z 313.194,A -85,B 0,C 180,E1 -16792.017,E2 -16792.017} C_VEL
LIN {X 0,Y 291.391,Z 313.236,A -85,B 0,C 180,E1 -16792.743,E2 -16792.743} C_VEL
LIN {X 0,Y 291.825,Z 316.254,A -85,B 0,C 180,E1 -16794.967,E2 -16794.967} C_VEL
LIN {X 0,Y 291.721,Z 319.813,A -85,B 0,C 180,E1 -16797.48,E2 -16797.48} C_VEL
LIN {X 0,Y 291.538,Z 325.274,A -85,B 0,C 180,E1 -16801.175,E2 -16801.175} C_VEL
LIN {X 0,Y 291.421,Z 331.14,A -85,B 0,C 180,E1 -16804.947,E2 -16804.947} C_VEL
LIN {X 0,Y 296.107,Z 345.762,A -85,B 0,C 180,E1 -16806.036,E2 -16806.036} C_VEL
LIN {X 0,Y 299.08,Z 357.96,A -85,B 0,C 180,E1 -16807.133,E2 -16807.133} C_VEL
LIN {X 0,Y 300.823,Z 368.326,A -85,B 0,C 180,E1 -16808.23,E2 -16808.23} C_VEL
LIN {X 0,Y 299.311,Z 380.607,A -85,B 0,C 180,E1 -16809.557,E2 -16809.557} C_VEL
LIN {X 0,Y 297.966,Z 390.351,A -85,B 0,C 180,E1 -16810.897,E2 -16810.897} C_VEL
LIN {X 0,Y 296.66,Z 399.324,A -85,B 0,C 180,E1 -16812.419,E2 -16812.419} C_VEL
LIN {X 0,Y 295.14,Z 407.527,A -85,B 0,C 180,E1 -16814.107,E2 -16814.107} C_VEL
LIN {X 0,Y 293.658,Z 415.524,A -85,B 0,C 180,E1 -16816.153,E2 -16816.153} C_VEL
LIN {X 0,Y 292.421,Z 421.951,A -85,B 0,C 180,E1 -16818.212,E2 -16818.212} C_VEL
LIN {X 0,Y 291.489,Z 427.055,A -85,B 0,C 180,E1 -16820.283,E2 -16820.283} C_VEL
LIN {X 0,Y 290.902,Z 430.562,A -85,B 0,C 180,E1 -16822.111,E2 -16822.111} C_VEL
LIN {X 0,Y 290.289,Z 433.911,A -85,B 0,C 180,E1 -16824.443,E2 -16824.443} C_VEL
LIN {X 0,Y 290.053,Z 435.319,A -85,B 0,C 180,E1 -16825.831,E2 -16825.831} C_VEL
LIN {X 0,Y 289.925,Z 436.305,A -85,B 0,C 180,E1 -16827.221,E2 -16827.221} C_VEL
LIN {X 0,Y 289.799,Z 437.145,A -85,B 0,C 180,E1 -16830,E2 -16830} C_VEL
LIN {X 0,Y 289.816,Z 436.953,A -85,B 0,C 180,E1 -16831.39,E2 -16831.39} C_VEL
LIN {X 0,Y 289.917,Z 436.368,A -85,B 0,C 180,E1 -16832.779,E2 -16832.779} C_VEL
LIN {X 0,Y 290.276,Z 434.047,A -85,B 0,C 180,E1 -16835.558,E2 -16835.558} C_VEL
LIN {X 0,Y 290.791,Z 431.04,A -85,B 0,C 180,E1 -16837.729,E2 -16837.729} C_VEL
LIN {X 0,Y 291.426,Z 427.304,A -85,B 0,C 180,E1 -16839.719,E2 -16839.719} C_VEL
LIN {X 0,Y 292.379,Z 422.265,A -85,B 0,C 180,E1 -16841.79,E2 -16841.79} C_VEL
LIN {X 0,Y 293.589,Z 415.904,A -85,B 0,C 180,E1 -16843.85,E2 -16843.85} C_VEL
LIN {X 0,Y 295.051,Z 407.992,A -85,B 0,C 180,E1 -16845.898,E2 -16845.898} C_VEL
LIN {X 0,Y 296.629,Z 399.891,A -85,B 0,C 180,E1 -16847.583,E2 -16847.583} C_VEL
LIN {X 0,Y 298.041,Z 389.947,A -85,B 0,C 180,E1 -16849.277,E2 -16849.277} C_VEL
LIN {X 0,Y 299.584,Z 378.727,A -85,B 0,C 180,E1 -16850.783,E2 -16850.783} C_VEL
LIN {X 0,Y 300.891,Z 367.706,A -85,B 0,C 180,E1 -16851.945,E2 -16851.945} C_VEL
LIN {X 0,Y 298.647,Z 355.842,A -85,B 0,C 180,E1 -16853.183,E2 -16853.183} C_VEL
LIN {X 0,Y 295.382,Z 343.279,A -85,B 0,C 180,E1 -16854.282,E2 -16854.282} C_VEL
LIN {X 0,Y 291.435,Z 331.12,A -85,B 0,C 180,E1 -16855.19,E2 -16855.19} C_VEL
LIN {X 0,Y 291.536,Z 325.487,A -85,B 0,C 180,E1 -16858.825,E2 -16858.825} C_VEL
LIN {X 0,Y 291.755,Z 320.019,A -85,B 0,C 180,E1 -16862.53,E2 -16862.53} C_VEL
LIN {X 0,Y 291.867,Z 316.431,A -85,B 0,C 180,E1 -16865.045,E2 -16865.045} C_VEL
LIN {X 0,Y 291.368,Z 313.192,A -85,B 0,C 180,E1 -16867.557,E2 -16867.557} C_VEL
LIN {X 0,Y 291.334,Z 313.198,A -85,B 0,C 180,E1 -16870.643,E2 -16870.643} C_VEL
LIN {X 0,Y 291.292,Z 313.204,A -85,B 0,C 180,E1 -16874.402,E2 -16874.402} C_VEL
LIN {X 0,Y 291.328,Z 313.194,A -85,B 0,C 180,E1 -16878.404,E2 -16878.404} C_VEL
LIN {X 0,Y 291.343,Z 313.191,A -85,B 0,C 180,E1 -16881.156,E2 -16881.156} C_VEL
LIN {X 0,Y 291.369,Z 313.191,A -85,B 0,C 180,E1 -16882.914,E2 -16882.914} C_VEL
LIN {X 0,Y 291.195,Z 313.249,A -85,B 0,C 180,E1 -16886.67,E2 -16886.67} C_VEL
LIN {X 0,Y 290.807,Z 319.681,A -85,B 0,C 180,E1 -16891.096,E2 -16891.096} C_VEL
LIN {X 0,Y 290.653,Z 325.353,A -85,B 0,C 180,E1 -16894.966,E2 -16894.966} C_VEL
LIN {X 0,Y 290.537,Z 331.266,A -85,B 0,C 180,E1 -16898.882,E2 -16898.882} C_VEL
LIN {X 0,Y 293.303,Z 346.535,A -85,B 0,C 180,E1 -16899.874,E2 -16899.874} C_VEL
LIN {X 0,Y 295.683,Z 359.925,A -85,B 0,C 180,E1 -16901.014,E2 -16901.014} C_VEL
LIN {X 0,Y 294.843,Z 371.899,A -85,B 0,C 180,E1 -16902.202,E2 -16902.202} C_VEL
LIN {X 0,Y 293.983,Z 383.617,A -85,B 0,C 180,E1 -16903.65,E2 -16903.65} C_VEL
LIN {X 0,Y 292.936,Z 388.356,A -85,B 0,C 180,E1 -16904.307,E2 -16904.307} C_VEL
LIN {X 0,Y 289.336,Z 395.687,A -85,B 0,C 180,E1 -16905.417,E2 -16905.417} C_VEL
LIN {X 0,Y 285.732,Z 402.606,A -85,B 0,C 180,E1 -16906.653,E2 -16906.653} C_VEL
LIN {X 0,Y 284.697,Z 406.621,A -85,B 0,C 180,E1 -16907.496,E2 -16907.496} C_VEL
LIN {X 0,Y 283.903,Z 415.405,A -85,B 0,C 180,E1 -16909.661,E2 -16909.661} C_VEL
LIN {X 0,Y 283.319,Z 422.395,A -85,B 0,C 180,E1 -16911.8,E2 -16911.8} C_VEL
LIN {X 0,Y 282.914,Z 428.84,A -85,B 0,C 180,E1 -16914.297,E2 -16914.297} C_VEL
LIN {X 0,Y 282.782,Z 433.029,A -85,B 0,C 180,E1 -16916.438,E2 -16916.438} C_VEL
LIN {X 0,Y 282.647,Z 436.127,A -85,B 0,C 180,E1 -16918.575,E2 -16918.575} C_VEL
LIN {X 0,Y 282.706,Z 437.626,A -85,B 0,C 180,E1 -16920,E2 -16920} C_VEL
LIN {X 0,Y 282.832,Z 438.702,A -85,B 0,C 180,E1 -16921.424,E2 -16921.424} C_VEL
LIN {X 0,Y 283.075,Z 439.309,A -85,B 0,C 180,E1 -16922.846,E2 -16922.846} C_VEL
LIN {X 0,Y 283.405,Z 439.514,A -85,B 0,C 180,E1 -16924.266,E2 -16924.266} C_VEL
LIN {X 0,Y 283.748,Z 439.306,A -85,B 0,C 180,E1 -16925.686,E2 -16925.686} C_VEL
LIN {X 0,Y 283.99,Z 438.669,A -85,B 0,C 180,E1 -16927.108,E2 -16927.108} C_VEL
LIN {X 0,Y 284.52,Z 437.615,A -85,B 0,C 180,E1 -16928.523,E2 -16928.523} C_VEL
LIN {X 0,Y 285.35,Z 436.127,A -85,B 0,C 180,E1 -16929.928,E2 -16929.928} C_VEL
LIN {X 0,Y 286.649,Z 433.034,A -85,B 0,C 180,E1 -16932.029,E2 -16932.029} C_VEL
LIN {X 0,Y 288.214,Z 428.92,A -85,B 0,C 180,E1 -16934.114,E2 -16934.114} C_VEL
LIN {X 0,Y 290.43,Z 422.628,A -85,B 0,C 180,E1 -16936.519,E2 -16936.519} C_VEL
LIN {X 0,Y 293.108,Z 414.596,A -85,B 0,C 180,E1 -16938.887,E2 -16938.887} C_VEL
LIN {X 0,Y 295.93,Z 405.946,A -85,B 0,C 180,E1 -16940.869,E2 -16940.869} C_VEL
LIN {X 0,Y 298.924,Z 395.435,A -85,B 0,C 180,E1 -16942.826,E2 -16942.826} C_VEL
LIN {X 0,Y 301.684,Z 384.947,A -85,B 0,C 180,E1 -16944.38,E2 -16944.38} C_VEL
LIN {X 0,Y 302.745,Z 380.687,A -85,B 0,C 180,E1 -16944.922,E2 -16944.922} C_VEL
LIN {X 0,Y 302.856,Z 377.773,A -85,B 0,C 180,E1 -16945.396,E2 -16945.396} C_VEL
LIN {X 0,Y 301.154,Z 368.73,A -85,B 0,C 180,E1 -16947.153,E2 -16947.153} C_VEL
LIN {X 0,Y 298.826,Z 360.814,A -85,B 0,C 180,E1 -16948.828,E2 -16948.828} C_VEL
LIN {X 0,Y 294.696,Z 350.237,A -85,B 0,C 180,E1 -16951.405,E2 -16951.405} C_VEL
LIN {X 0,Y 292.448,Z 345.62,A -85,B 0,C 180,E1 -16952.742,E2 -16952.742} C_VEL
LIN {X 0,Y 290.638,Z 341.957,A -85,B 0,C 180,E1 -16953.899,E2 -16953.899} C_VEL
LIN {X 0,Y 290.565,Z 341.557,A -85,B 0,C 180,E1 -16954.076,E2 -16954.076} C_VEL
LIN {X 0,Y 291.017,Z 339.328,A -85,B 0,C 180,E1 -16957.161,E2 -16957.161} C_VEL
LIN {X 0,Y 291.253,Z 337.724,A -85,B 0,C 180,E1 -16960.656,E2 -16960.656} C_VEL
LIN {X 0,Y 291.189,Z 337.33,A -85,B 0,C 180,E1 -16963.609,E2 -16963.609} C_VEL
LIN {X 0,Y 290.875,Z 338.01,A -85,B 0,C 180,E1 -16966.456,E2 -16966.456} C_VEL
LIN {X 0,Y 290.809,Z 339.614,A -85,B 0,C 180,E1 -16969.269,E2 -16969.269} C_VEL
LIN {X 0,Y 290.756,Z 342.366,A -85,B 0,C 180,E1 -16971.948,E2 -16971.948} C_VEL
LIN {X 0,Y 290.249,Z 345.02,A -85,B 0,C 180,E1 -16973.569,E2 -16973.569} C_VEL
LIN {X 0,Y 289.494,Z 350.704,A -85,B 0,C 180,E1 -16976.206,E2 -16976.206} C_VEL
LIN {X 0,Y 292.839,Z 361.073,A -85,B 0,C 180,E1 -16978.508,E2 -16978.508} C_VEL
LIN {X 0,Y 294.969,Z 370.593,A -85,B 0,C 180,E1 -16980.122,E2 -16980.122} C_VEL
LIN {X 0,Y 296.571,Z 381.803,A -85,B 0,C 180,E1 -16981.813,E2 -16981.813} C_VEL
LIN {X 0,Y 297.268,Z 394.653,A -85,B 0,C 180,E1 -16983.656,E2 -16983.656} C_VEL
LIN {X 0,Y 296.32,Z 406.267,A -85,B 0,C 180,E1 -16985.266,E2 -16985.266} C_VEL
LIN {X 0,Y 294.952,Z 418.516,A -85,B 0,C 180,E1 -16987.22,E2 -16987.22} C_VEL
LIN {X 0,Y 291.861,Z 429.948,A -85,B 0,C 180,E1 -16989.195,E2 -16989.195} C_VEL
LIN {X 0,Y 289.286,Z 439.353,A -85,B 0,C 180,E1 -16991.222,E2 -16991.222} C_VEL
LIN {X 0,Y 286.905,Z 448.36,A -85,B 0,C 180,E1 -16993.638,E2 -16993.638} C_VEL
LIN {X 0,Y 285.29,Z 454.648,A -85,B 0,C 180,E1 -16995.739,E2 -16995.739} C_VEL
LIN {X 0,Y 284.067,Z 459.784,A -85,B 0,C 180,E1 -16997.86,E2 -16997.86} C_VEL
LIN {X 0,Y 283.066,Z 465.012,A -85,B 0,C 180,E1 -17000.713,E2 -17000.713} C_VEL
LIN {X 0,Y 282.694,Z 467.809,A -85,B 0,C 180,E1 -17002.859,E2 -17002.859} C_VEL
LIN {X 0,Y 282.543,Z 469.178,A -85,B 0,C 180,E1 -17004.29,E2 -17004.29} C_VEL
LIN {X 0,Y 282.542,Z 470.104,A -85,B 0,C 180,E1 -17005.72,E2 -17005.72} C_VEL
LIN {X 0,Y 282.537,Z 470.624,A -85,B 0,C 180,E1 -17007.148,E2 -17007.148} C_VEL
LIN {X 0,Y 282.862,Z 470.673,A -85,B 0,C 180,E1 -17010,E2 -17010} C_VEL
LIN {X 0,Y 282.679,Z 470.435,A -85,B 0,C 180,E1 -17011.425,E2 -17011.425} C_VEL
LIN {X 0,Y 282.579,Z 468.773,A -85,B 0,C 180,E1 -17014.279,E2 -17014.279} C_VEL
LIN {X 0,Y 282.641,Z 467.018,A -85,B 0,C 180,E1 -17015.944,E2 -17015.944} C_VEL
LIN {X 0,Y 282.885,Z 463.035,A -85,B 0,C 180,E1 -17018.573,E2 -17018.573} C_VEL
LIN {X 0,Y 284.216,Z 454.24,A -85,B 0,C 180,E1 -17022.859,E2 -17022.859} C_VEL
LIN {X 0,Y 285.893,Z 447.686,A -85,B 0,C 180,E1 -17025.323,E2 -17025.323} C_VEL
LIN {X 0,Y 287.82,Z 439.621,A -85,B 0,C 180,E1 -17027.767,E2 -17027.767} C_VEL
LIN {X 0,Y 290.159,Z 431.196,A -85,B 0,C 180,E1 -17029.822,E2 -17029.822} C_VEL
LIN {X 0,Y 292.97,Z 421.14,A -85,B 0,C 180,E1 -17031.828,E2 -17031.828} C_VEL
LIN {X 0,Y 294.193,Z 415.464,A -85,B 0,C 180,E1 -17032.843,E2 -17032.843} C_VEL
LIN {X 0,Y 295.664,Z 404.642,A -85,B 0,C 180,E1 -17034.645,E2 -17034.645} C_VEL
LIN {X 0,Y 296.407,Z 395.633,A -85,B 0,C 180,E1 -17036.017,E2 -17036.017} C_VEL
LIN {X 0,Y 296.156,Z 385.343,A -85,B 0,C 180,E1 -17037.605,E2 -17037.605} C_VEL
LIN {X 0,Y 294.969,Z 375.137,A -85,B 0,C 180,E1 -17039.254,E2 -17039.254} C_VEL
LIN {X 0,Y 292.741,Z 364.256,A -85,B 0,C 180,E1 -17041.201,E2 -17041.201} C_VEL
LIN {X 0,Y 291.788,Z 360.061,A -85,B 0,C 180,E1 -17041.998,E2 -17041.998} C_VEL
LIN {X 0,Y 290.599,Z 356.281,A -85,B 0,C 180,E1 -17042.817,E2 -17042.817} C_VEL
LIN {X 0,Y 290.061,Z 353.943,A -85,B 0,C 180,E1 -17043.29,E2 -17043.29} C_VEL
LIN {X 0,Y 288.767,Z 350.511,A -85,B 0,C 180,E1 -17044.158,E2 -17044.158} C_VEL
LIN {X 0,Y 288.327,Z 347.531,A -85,B 0,C 180,E1 -17044.771,E2 -17044.771} C_VEL
LIN {X 0,Y 289.497,Z 343.856,A -85,B 0,C 180,E1 -17047.367,E2 -17047.367} C_VEL
LIN {X 0,Y 289.568,Z 341.725,A -85,B 0,C 180,E1 -17049.127,E2 -17049.127} C_VEL
LIN {X 0,Y 289.268,Z 339.611,A -85,B 0,C 180,E1 -17051.134,E2 -17051.134} C_VEL
LIN {X 0,Y 288.696,Z 336.276,A -85,B 0,C 180,E1 -17054.909,E2 -17054.909} C_VEL
LIN {X 0,Y 288.187,Z 333.523,A -85,B 0,C 180,E1 -17059.113,E2 -17059.113} C_VEL
LIN {X 0,Y 287.873,Z 332.047,A -85,B 0,C 180,E1 -17062.386,E2 -17062.386} C_VEL
LIN {X 0,Y 287.713,Z 331.321,A -85,B 0,C 180,E1 -17064.808,E2 -17064.808} C_VEL
LIN {X 0,Y 289.304,Z 334.059,A -85,B 0,C 180,E1 -17066.032,E2 -17066.032} C_VEL
LIN {X 0,Y 290.24,Z 334.777,A -85,B 0,C 180,E1 -17066.568,E2 -17066.568} C_VEL
LIN {X 0,Y 293.647,Z 338.947,A -85,B 0,C 180,E1 -17068.522,E2 -17068.522} C_VEL
LIN {X 0,Y 297.882,Z 345.243,A -85,B 0,C 180,E1 -17070.804,E2 -17070.804} C_VEL
LIN {X 0,Y 301.589,Z 352.593,A -85,B 0,C 180,E1 -17072.922,E2 -17072.922} C_VEL
LIN {X 0,Y 304.161,Z 360.273,A -85,B 0,C 180,E1 -17074.78,E2 -17074.78} C_VEL
LIN {X 0,Y 304.348,Z 362.411,A -85,B 0,C 180,E1 -17075.203,E2 -17075.203} C_VEL
LIN {X 0,Y 301.664,Z 372.795,A -85,B 0,C 180,E1 -17076.668,E2 -17076.668} C_VEL
LIN {X 0,Y 299.019,Z 382.064,A -85,B 0,C 180,E1 -17078.273,E2 -17078.273} C_VEL
LIN {X 0,Y 296.134,Z 391.233,A -85,B 0,C 180,E1 -17080.233,E2 -17080.233} C_VEL
LIN {X 0,Y 293.584,Z 398.753,A -85,B 0,C 180,E1 -17082.229,E2 -17082.229} C_VEL
LIN {X 0,Y 290.978,Z 405.705,A -85,B 0,C 180,E1 -17084.592,E2 -17084.592} C_VEL
LIN {X 0,Y 289.161,Z 410.242,A -85,B 0,C 180,E1 -17086.579,E2 -17086.579} C_VEL
LIN {X 0,Y 287.448,Z 413.96,A -85,B 0,C 180,E1 -17088.72,E2 -17088.72} C_VEL
LIN {X 0,Y 286.534,Z 415.819,A -85,B 0,C 180,E1 -17090.114,E2 -17090.114} C_VEL
LIN {X 0,Y 285.753,Z 417.19,A -85,B 0,C 180,E1 -17091.514,E2 -17091.514} C_VEL
LIN {X 0,Y 285.104,Z 418.15,A -85,B 0,C 180,E1 -17092.92,E2 -17092.92} C_VEL
LIN {X 0,Y 284.537,Z 418.715,A -85,B 0,C 180,E1 -17094.33,E2 -17094.33} C_VEL
LIN {X 0,Y 284.031,Z 418.857,A -85,B 0,C 180,E1 -17095.743,E2 -17095.743} C_VEL
LIN {X 0,Y 283.652,Z 418.569,A -85,B 0,C 180,E1 -17097.16,E2 -17097.16} C_VEL
LIN {X 0,Y 283.353,Z 417.877,A -85,B 0,C 180,E1 -17098.579,E2 -17098.579} C_VEL
LIN {X 0,Y 283.221,Z 416.767,A -85,B 0,C 180,E1 -17100,E2 -17100} C_VEL
LIN {X 0,Y 283.22,Z 415.192,A -85,B 0,C 180,E1 -17101.422,E2 -17101.422} C_VEL
LIN {X 0,Y 283.365,Z 412.038,A -85,B 0,C 180,E1 -17103.555,E2 -17103.555} C_VEL
LIN {X 0,Y 283.586,Z 407.809,A -85,B 0,C 180,E1 -17105.689,E2 -17105.689} C_VEL
LIN {X 0,Y 283.827,Z 402.152,A -85,B 0,C 180,E1 -17107.917,E2 -17107.917} C_VEL
LIN {X 0,Y 284.348,Z 395.688,A -85,B 0,C 180,E1 -17109.963,E2 -17109.963} C_VEL
LIN {X 0,Y 285.091,Z 387.413,A -85,B 0,C 180,E1 -17112.096,E2 -17112.096} C_VEL
LIN {X 0,Y 286.02,Z 377.211,A -85,B 0,C 180,E1 -17114.224,E2 -17114.224} C_VEL
LIN {X 0,Y 287.1,Z 366.776,A -85,B 0,C 180,E1 -17115.985,E2 -17115.985} C_VEL
LIN {X 0,Y 288.137,Z 354.505,A -85,B 0,C 180,E1 -17117.665,E2 -17117.665} C_VEL
LIN {X 0,Y 289.006,Z 342.47,A -85,B 0,C 180,E1 -17118.981,E2 -17118.981} C_VEL
LIN {X 0,Y 289.22,Z 336.708,A -85,B 0,C 180,E1 -17119.519,E2 -17119.519} C_VEL
LIN {X 0,Y 286.666,Z 325.078,A -85,B 0,C 180,E1 -17120.56,E2 -17120.56} C_VEL
LIN {X 0,Y 283.983,Z 314.1,A -85,B 0,C 180,E1 -17121.372,E2 -17121.372} C_VEL
LIN {X 0,Y 284.186,Z 314.083,A -85,B 0,C 180,E1 -17124.861,E2 -17124.861} C_VEL
LIN {X 0,Y 284.294,Z 314.068,A -85,B 0,C 180,E1 -17128.015,E2 -17128.015} C_VEL
LIN {X 0,Y 284.295,Z 314.063,A -85,B 0,C 180,E1 -17131.275,E2 -17131.275} C_VEL
LIN {X 0,Y 284.363,Z 314.056,A -85,B 0,C 180,E1 -17135.354,E2 -17135.354} C_VEL
LIN {X 0,Y 284.325,Z 314.069,A -85,B 0,C 180,E1 -17138.167,E2 -17138.167} C_VEL
LIN {X 0,Y 284.271,Z 314.075,A -85,B 0,C 180,E1 -17142.124,E2 -17142.124} C_VEL
LIN {X 0,Y 284.257,Z 314.076,A -85,B 0,C 180,E1 -17146.189,E2 -17146.189} C_VEL
LIN {X 0,Y 284.308,Z 314.071,A -85,B 0,C 180,E1 -17150.024,E2 -17150.024} C_VEL
LIN {X 0,Y 284.333,Z 314.152,A -85,B 0,C 180,E1 -17152.276,E2 -17152.276} C_VEL
LIN {X 0,Y 284.876,Z 318.392,A -85,B 0,C 180,E1 -17155.429,E2 -17155.429} C_VEL
LIN {X 0,Y 284.693,Z 323.149,A -85,B 0,C 180,E1 -17158.774,E2 -17158.774} C_VEL
LIN {X 0,Y 284.528,Z 329.137,A -85,B 0,C 180,E1 -17162.776,E2 -17162.776} C_VEL
LIN {X 0,Y 284.494,Z 331.502,A -85,B 0,C 180,E1 -17164.297,E2 -17164.297} C_VEL
LIN {X 0,Y 289.165,Z 345.876,A -85,B 0,C 180,E1 -17165.407,E2 -17165.407} C_VEL
LIN {X 0,Y 292.147,Z 357.845,A -85,B 0,C 180,E1 -17166.514,E2 -17166.514} C_VEL
LIN {X 0,Y 294.115,Z 368.734,A -85,B 0,C 180,E1 -17167.707,E2 -17167.707} C_VEL
LIN {X 0,Y 292.85,Z 379.633,A -85,B 0,C 180,E1 -17168.901,E2 -17168.901} C_VEL
LIN {X 0,Y 291.316,Z 390.475,A -85,B 0,C 180,E1 -17170.398,E2 -17170.398} C_VEL
LIN {X 0,Y 289.928,Z 399.734,A -85,B 0,C 180,E1 -17171.997,E2 -17171.997} C_VEL
LIN {X 0,Y 288.34,Z 407.939,A -85,B 0,C 180,E1 -17173.722,E2 -17173.722} C_VEL
LIN {X 0,Y 286.773,Z 415.938,A -85,B 0,C 180,E1 -17175.814,E2 -17175.814} C_VEL
LIN {X 0,Y 285.495,Z 422.365,A -85,B 0,C 180,E1 -17177.922,E2 -17177.922} C_VEL
LIN {X 0,Y 284.495,Z 427.47,A -85,B 0,C 180,E1 -17180.042,E2 -17180.042} C_VEL
LIN {X 0,Y 283.842,Z 431.226,A -85,B 0,C 180,E1 -17182.061,E2 -17182.061} C_VEL
LIN {X 0,Y 283.251,Z 434.325,A -85,B 0,C 180,E1 -17184.304,E2 -17184.304} C_VEL
LIN {X 0,Y 282.989,Z 435.734,A -85,B 0,C 180,E1 -17185.727,E2 -17185.727} C_VEL
LIN {X 0,Y 282.731,Z 437.33,A -85,B 0,C 180,E1 -17188.576,E2 -17188.576} C_VEL
LIN {X 0,Y 282.712,Z 437.56,A -85,B 0,C 180,E1 -17190,E2 -17190} C_VEL
LIN {X 0,Y 282.731,Z 437.367,A -85,B 0,C 180,E1 -17191.424,E2 -17191.424} C_VEL
LIN {X 0,Y 282.834,Z 436.782,A -85,B 0,C 180,E1 -17192.849,E2 -17192.849} C_VEL
LIN {X 0,Y 283.239,Z 434.46,A -85,B 0,C 180,E1 -17195.696,E2 -17195.696} C_VEL
LIN {X 0,Y 283.72,Z 431.706,A -85,B 0,C 180,E1 -17197.761,E2 -17197.761} C_VEL
LIN {X 0,Y 284.447,Z 427.716,A -85,B 0,C 180,E1 -17199.96,E2 -17199.96} C_VEL
LIN {X 0,Y 285.459,Z 422.675,A -85,B 0,C 180,E1 -17202.08,E2 -17202.08} C_VEL
LIN {X 0,Y 286.715,Z 416.313,A -85,B 0,C 180,E1 -17204.189,E2 -17204.189} C_VEL
LIN {X 0,Y 288.251,Z 408.399,A -85,B 0,C 180,E1 -17206.283,E2 -17206.283} C_VEL
LIN {X 0,Y 289.899,Z 400.294,A -85,B 0,C 180,E1 -17208.005,E2 -17208.005} C_VEL
LIN {X 0,Y 291.367,Z 390.347,A -85,B 0,C 180,E1 -17209.736,E2 -17209.736} C_VEL
LIN {X 0,Y 292.984,Z 379.121,A -85,B 0,C 180,E1 -17211.273,E2 -17211.273} C_VEL
LIN {X 0,Y 294.224,Z 369.794,A -85,B 0,C 180,E1 -17212.284,E2 -17212.284} C_VEL
LIN {X 0,Y 292.503,Z 359.474,A -85,B 0,C 180,E1 -17213.431,E2 -17213.431} C_VEL
LIN {X 0,Y 289.577,Z 347.273,A -85,B 0,C 180,E1 -17214.594,E2 -17214.594} C_VEL
LIN {X 0,Y 285.443,Z 334.462,A -85,B 0,C 180,E1 -17215.611,E2 -17215.611} C_VEL
LIN {X 0,Y 284.496,Z 331.534,A -85,B 0,C 180,E1 -17215.829,E2 -17215.829} C_VEL
LIN {X 0,Y 284.672,Z 324.82,A -85,B 0,C 180,E1 -17220.221,E2 -17220.221} C_VEL
LIN {X 0,Y 284.991,Z 318.584,A -85,B 0,C 180,E1 -17224.555,E2 -17224.555} C_VEL
LIN {X 0,Y 284.331,Z 314.123,A -85,B 0,C 180,E1 -17227.883,E2 -17227.883} C_VEL
LIN {X 0,Y 284.274,Z 314.076,A -85,B 0,C 180,E1 -17231.875,E2 -17231.875} C_VEL
LIN {X 0,Y 284.257,Z 314.076,A -85,B 0,C 180,E1 -17236.189,E2 -17236.189} C_VEL
LIN {X 0,Y 284.308,Z 314.072,A -85,B 0,C 180,E1 -17240.024,E2 -17240.024} C_VEL
LIN {X 0,Y 284.276,Z 314.076,A -85,B 0,C 180,E1 -17243.605,E2 -17243.605} C_VEL
LIN {X 0,Y 284.177,Z 314.117,A -85,B 0,C 180,E1 -17246.614,E2 -17246.614} C_VEL
LIN {X 0,Y 283.773,Z 320.634,A -85,B 0,C 180,E1 -17251.122,E2 -17251.122} C_VEL
LIN {X 0,Y 283.596,Z 326.39,A -85,B 0,C 180,E1 -17255.084,E2 -17255.084} C_VEL
LIN {X 0,Y 283.478,Z 331.609,A -85,B 0,C 180,E1 -17258.62,E2 -17258.62} C_VEL
LIN {X 0,Y 286,Z 345.683,A -85,B 0,C 180,E1 -17259.531,E2 -17259.531} C_VEL
LIN {X 0,Y 288.604,Z 360.371,A -85,B 0,C 180,E1 -17260.807,E2 -17260.807} C_VEL
LIN {X 0,Y 287.833,Z 372.183,A -85,B 0,C 180,E1 -17262.01,E2 -17262.01} C_VEL
LIN {X 0,Y 286.97,Z 383.707,A -85,B 0,C 180,E1 -17263.459,E2 -17263.459} C_VEL
LIN {X 0,Y 285.825,Z 395.01,A -85,B 0,C 180,E1 -17265.22,E2 -17265.22} C_VEL
LIN {X 0,Y 284.821,Z 405.131,A -85,B 0,C 180,E1 -17267.169,E2 -17267.169} C_VEL
LIN {X 0,Y 284.697,Z 406.621,A -85,B 0,C 180,E1 -17267.496,E2 -17267.496} C_VEL
LIN {X 0,Y 283.714,Z 410.501,A -85,B 0,C 180,E1 -17268.373,E2 -17268.373} C_VEL
LIN {X 0,Y 280.336,Z 416.368,A -85,B 0,C 180,E1 -17269.848,E2 -17269.848} C_VEL
LIN {X 0,Y 276.989,Z 421.631,A -85,B 0,C 180,E1 -17271.445,E2 -17271.445} C_VEL
LIN {X 0,Y 276.081,Z 424.571,A -85,B 0,C 180,E1 -17272.496,E2 -17272.496} C_VEL
LIN {X 0,Y 275.805,Z 430.221,A -85,B 0,C 180,E1 -17274.883,E2 -17274.883} C_VEL
LIN {X 0,Y 275.639,Z 434.193,A -85,B 0,C 180,E1 -17277.077,E2 -17277.077} C_VEL
LIN {X 0,Y 275.561,Z 436.259,A -85,B 0,C 180,E1 -17278.538,E2 -17278.538} C_VEL
LIN {X 0,Y 275.613,Z 437.838,A -85,B 0,C 180,E1 -17280,E2 -17280} C_VEL
LIN {X 0,Y 275.742,Z 439.014,A -85,B 0,C 180,E1 -17281.46,E2 -17281.46} C_VEL
LIN {X 0,Y 275.997,Z 439.75,A -85,B 0,C 180,E1 -17282.919,E2 -17282.919} C_VEL
LIN {X 0,Y 276.34,Z 440.032,A -85,B 0,C 180,E1 -17284.376,E2 -17284.376} C_VEL
LIN {X 0,Y 276.694,Z 439.924,A -85,B 0,C 180,E1 -17285.831,E2 -17285.831} C_VEL
LIN {X 0,Y 276.98,Z 439.424,A -85,B 0,C 180,E1 -17287.289,E2 -17287.289} C_VEL
LIN {X 0,Y 278.335,Z 437.228,A -85,B 0,C 180,E1 -17290.015,E2 -17290.015} C_VEL
LIN {X 0,Y 279.825,Z 434.177,A -85,B 0,C 180,E1 -17292.327,E2 -17292.327} C_VEL
LIN {X 0,Y 281.467,Z 430.254,A -85,B 0,C 180,E1 -17294.459,E2 -17294.459} C_VEL
LIN {X 0,Y 283.44,Z 425.256,A -85,B 0,C 180,E1 -17296.568,E2 -17296.568} C_VEL
LIN {X 0,Y 286.233,Z 417.775,A -85,B 0,C 180,E1 -17298.986,E2 -17298.986} C_VEL
LIN {X 0,Y 289.089,Z 409.835,A -85,B 0,C 180,E1 -17301.013,E2 -17301.013} C_VEL
LIN {X 0,Y 292.219,Z 400.092,A -85,B 0,C 180,E1 -17303.006,E2 -17303.006} C_VEL
LIN {X 0,Y 295.274,Z 389.767,A -85,B 0,C 180,E1 -17304.716,E2 -17304.716} C_VEL
LIN {X 0,Y 297.267,Z 382.525,A -85,B 0,C 180,E1 -17305.718,E2 -17305.718} C_VEL
LIN {X 0,Y 296.839,Z 377.313,A -85,B 0,C 180,E1 -17306.734,E2 -17306.734} C_VEL
LIN {X 0,Y 295.257,Z 369.454,A -85,B 0,C 180,E1 -17308.428,E2 -17308.428} C_VEL
LIN {X 0,Y 292.955,Z 361.778,A -85,B 0,C 180,E1 -17310.272,E2 -17310.272} C_VEL
LIN {X 0,Y 290.328,Z 354.76,A -85,B 0,C 180,E1 -17312.178,E2 -17312.178} C_VEL
LIN {X 0,Y 288.96,Z 351.315,A -85,B 0,C 180,E1 -17313.218,E2 -17313.218} C_VEL
LIN {X 0,Y 286.93,Z 347.115,A -85,B 0,C 180,E1 -17314.708,E2 -17314.708} C_VEL
LIN {X 0,Y 284.589,Z 342.958,A -85,B 0,C 180,E1 -17316.581,E2 -17316.581} C_VEL
LIN {X 0,Y 284.958,Z 341.376,A -85,B 0,C 180,E1 -17319.885,E2 -17319.885} C_VEL
LIN {X 0,Y 285.098,Z 340.918,A -85,B 0,C 180,E1 -17322.308,E2 -17322.308} C_VEL
LIN {X 0,Y 285.03,Z 341.048,A -85,B 0,C 180,E1 -17324.352,E2 -17324.352} C_VEL
LIN {X 0,Y 284.8,Z 342.497,A -85,B 0,C 180,E1 -17327.758,E2 -17327.758} C_VEL
LIN {X 0,Y 284.874,Z 344.337,A -85,B 0,C 180,E1 -17330.101,E2 -17330.101} C_VEL
LIN {X 0,Y 284.754,Z 346.835,A -85,B 0,C 180,E1 -17332.166,E2 -17332.166} C_VEL
LIN {X 0,Y 284.253,Z 350.108,A -85,B 0,C 180,E1 -17333.904,E2 -17333.904} C_VEL
LIN {X 0,Y 286.317,Z 357.408,A -85,B 0,C 180,E1 -17335.883,E2 -17335.883} C_VEL
LIN {X 0,Y 288.885,Z 366.153,A -85,B 0,C 180,E1 -17337.896,E2 -17337.896} C_VEL
LIN {X 0,Y 290.382,Z 374.809,A -85,B 0,C 180,E1 -17339.452,E2 -17339.452} C_VEL
LIN {X 0,Y 291.45,Z 385.413,A -85,B 0,C 180,E1 -17341.166,E2 -17341.166} C_VEL
LIN {X 0,Y 291.625,Z 397.915,A -85,B 0,C 180,E1 -17343.086,E2 -17343.086} C_VEL
LIN {X 0,Y 289.837,Z 412.365,A -85,B 0,C 180,E1 -17345.274,E2 -17345.274} C_VEL
LIN {X 0,Y 288.636,Z 420.441,A -85,B 0,C 180,E1 -17346.692,E2 -17346.692} C_VEL
